// TIA Portal V20 export
FUNCTION "ParameterMove" : Void   // FC22, LAD
// stored: SetENOAutomatically false
   VAR_TEMP
      tempSoftCamDRApplyLoop : Array[1..41] of Int;
      tempSoftCamDRReadLoop : Array[1..41] of Int;
      tempButtonRisingEdge : "HMI_IF_Parameter_Save Button_UDT";
   END_VAR
   VAR_TEMP   // added for the SCL form of the ladder/FBD networks
      _w1 : Bool;
      _w2 : Bool;
      _w3 : Bool;
   END_VAR
BEGIN

REGION Network 2 (SCL): Button Rising Edge
   #tempButtonRisingEdge.Read := "HMI_Interface_Parameter"."Save Button".Read AND NOT "HMI_Interface_Parameter"."Save Button Old".Read;
   #tempButtonRisingEdge.Save := "HMI_Interface_Parameter"."Save Button".Save AND NOT "HMI_Interface_Parameter"."Save Button Old".Save;
   #tempButtonRisingEdge.Apply := "HMI_Interface_Parameter"."Save Button".Apply AND NOT "HMI_Interface_Parameter"."Save Button Old".Apply;
   "HMI_Interface_Parameter"."Save Button Old".Read := "HMI_Interface_Parameter"."Save Button".Read;
   "HMI_Interface_Parameter"."Save Button Old".Save := "HMI_Interface_Parameter"."Save Button".Save;
   "HMI_Interface_Parameter"."Save Button Old".Apply := "HMI_Interface_Parameter"."Save Button".Apply;
END_REGION

REGION Network 3 (SCL): HMI Parameter Text Set Value
   IF #tempButtonRisingEdge.Apply THEN
       "HMI_Interface_Parameter".Parameter_Text[0]."Process Value" := "HMI_Interface_Parameter".Parameter_Text[0]."Set Value";
       "HMI_Interface_Parameter".Parameter_Text[2]."Process Value" := "HMI_Interface_Parameter".Parameter_Text[2]."Set Value";
       "HMI_Interface_Parameter".Parameter_Text[6]."Process Value" := "HMI_Interface_Parameter".Parameter_Text[6]."Set Value";
       "HMI_Interface_Parameter".Parameter_Text[7]."Process Value" := "HMI_Interface_Parameter".Parameter_Text[7]."Set Value";
       "HMI_Interface_Parameter".Parameter_Text[9]."Process Value" := "HMI_Interface_Parameter".Parameter_Text[9]."Set Value";
       "HMI_Interface_Parameter".Parameter_Text[10]."Process Value" := "HMI_Interface_Parameter".Parameter_Text[10]."Set Value";
       "HMI_Interface_Parameter".Parameter_Text[11]."Process Value" := "HMI_Interface_Parameter".Parameter_Text[11]."Set Value";
       "HMI_Interface_Parameter".Parameter_Text[13]."Process Value" := "HMI_Interface_Parameter".Parameter_Text[13]."Set Value";
       "HMI_Interface_Parameter".Parameter_Text[14]."Process Value" := "HMI_Interface_Parameter".Parameter_Text[14]."Set Value";
       "HMI_Interface_Parameter".Parameter_Text[15]."Process Value" := "HMI_Interface_Parameter".Parameter_Text[15]."Set Value";
       "HMI_Interface_Parameter".Parameter_Text[16]."Process Value" := "HMI_Interface_Parameter".Parameter_Text[16]."Set Value";
       "HMI_Interface_Parameter".Parameter_Text[17]."Process Value" := "HMI_Interface_Parameter".Parameter_Text[17]."Set Value";
       "HMI_Interface_Parameter".Parameter_Text[18]."Process Value" := "HMI_Interface_Parameter".Parameter_Text[18]."Set Value";
       "HMI_Interface_Parameter".Parameter_Text[19]."Process Value" := "HMI_Interface_Parameter".Parameter_Text[19]."Set Value";
       "HMI_Interface_Parameter".Parameter_Text[20]."Process Value" := "HMI_Interface_Parameter".Parameter_Text[20]."Set Value";
       "HMI_Interface_Parameter".Parameter_Text[21]."Process Value" := "HMI_Interface_Parameter".Parameter_Text[21]."Set Value";
       "HMI_Interface_Parameter".Parameter_Text[22]."Process Value" := "HMI_Interface_Parameter".Parameter_Text[22]."Set Value";
       "HMI_Interface_Parameter".Parameter_Text[23]."Process Value" := "HMI_Interface_Parameter".Parameter_Text[23]."Set Value";
       "HMI_Interface_Parameter".Parameter_Text[24]."Process Value" := "HMI_Interface_Parameter".Parameter_Text[24]."Set Value";
       "HMI_Interface_Parameter".Parameter_Text[25]."Process Value" := "HMI_Interface_Parameter".Parameter_Text[25]."Set Value";
       "HMI_Interface_Parameter".Parameter_Text[26]."Process Value" := "HMI_Interface_Parameter".Parameter_Text[26]."Set Value";
       "HMI_Interface_Parameter".Parameter_Text[27]."Process Value" := "HMI_Interface_Parameter".Parameter_Text[27]."Set Value";
       "HMI_Interface_Parameter".Parameter_Text[28]."Process Value" := "HMI_Interface_Parameter".Parameter_Text[28]."Set Value";
       "HMI_Interface_Parameter".Parameter_Text[29]."Process Value" := "HMI_Interface_Parameter".Parameter_Text[29]."Set Value";
       "HMI_Interface_Parameter".Parameter_Text[30]."Process Value" := "HMI_Interface_Parameter".Parameter_Text[30]."Set Value";
       "HMI_Interface_Parameter".Parameter_Text[31]."Process Value" := "HMI_Interface_Parameter".Parameter_Text[31]."Set Value";
       "HMI_Interface_Parameter".Parameter_Text[32]."Process Value" := "HMI_Interface_Parameter".Parameter_Text[32]."Set Value";
       "HMI_Interface_Parameter".Parameter_Text[33]."Process Value" := "HMI_Interface_Parameter".Parameter_Text[33]."Set Value";
       "HMI_Interface_Parameter".Parameter_Text[34]."Process Value" := "HMI_Interface_Parameter".Parameter_Text[34]."Set Value";
       "HMI_Interface_Parameter".Parameter_Text[35]."Process Value" := "HMI_Interface_Parameter".Parameter_Text[35]."Set Value";
       "HMI_Interface_Parameter".Parameter_Text[36]."Process Value" := "HMI_Interface_Parameter".Parameter_Text[36]."Set Value";
       "HMI_Interface_Parameter".Parameter_Text[37]."Process Value" := "HMI_Interface_Parameter".Parameter_Text[37]."Set Value";
       "HMI_Interface_Parameter".Parameter_Text[38]."Process Value" := "HMI_Interface_Parameter".Parameter_Text[38]."Set Value";
       "HMI_Interface_Parameter".Parameter_Text[39]."Process Value" := "HMI_Interface_Parameter".Parameter_Text[39]."Set Value";
       "HMI_Interface_Parameter".Parameter_Text[40]."Process Value" := "HMI_Interface_Parameter".Parameter_Text[40]."Set Value";
       "HMI_Interface_Parameter".Parameter_Text[41]."Process Value" := "HMI_Interface_Parameter".Parameter_Text[41]."Set Value";
       "HMI_Interface_Parameter".Parameter_Text[42]."Process Value" := "HMI_Interface_Parameter".Parameter_Text[42]."Set Value";
       "HMI_Interface_Parameter".Parameter_Text[43]."Process Value" := "HMI_Interface_Parameter".Parameter_Text[43]."Set Value";
       "HMI_Interface_Parameter".Parameter_Text[44]."Process Value" := "HMI_Interface_Parameter".Parameter_Text[44]."Set Value";
       "HMI_Interface_Parameter".Parameter_Text[45]."Process Value" := "HMI_Interface_Parameter".Parameter_Text[45]."Set Value";
       "HMI_Interface_Parameter".Parameter_Text[46]."Process Value" := "HMI_Interface_Parameter".Parameter_Text[46]."Set Value";
       "HMI_Interface_Parameter".Parameter_Text[47]."Process Value" := "HMI_Interface_Parameter".Parameter_Text[47]."Set Value";
       "HMI_Interface_Parameter".Parameter_Text[48]."Process Value" := "HMI_Interface_Parameter".Parameter_Text[48]."Set Value";
       "HMI_Interface_Parameter".Parameter_Text[49]."Process Value" := "HMI_Interface_Parameter".Parameter_Text[49]."Set Value";
       "HMI_Interface_Parameter".Parameter_Text[50]."Process Value" := "HMI_Interface_Parameter".Parameter_Text[50]."Set Value";
       "HMI_Interface_Parameter".Parameter_Text[51]."Process Value" := "HMI_Interface_Parameter".Parameter_Text[51]."Set Value";
       "HMI_Interface_Parameter".Parameter_Text[52]."Process Value" := "HMI_Interface_Parameter".Parameter_Text[52]."Set Value";
       "HMI_Interface_Parameter".Parameter_Text[53]."Process Value" := "HMI_Interface_Parameter".Parameter_Text[53]."Set Value";
       "HMI_Interface_Parameter".Parameter_Text[54]."Process Value" := "HMI_Interface_Parameter".Parameter_Text[54]."Set Value";
       "HMI_Interface_Parameter".Parameter_Text[55]."Process Value" := "HMI_Interface_Parameter".Parameter_Text[55]."Set Value";
       "HMI_Interface_Parameter".Parameter_Text[56]."Process Value" := "HMI_Interface_Parameter".Parameter_Text[56]."Set Value";
       "HMI_Interface_Parameter".Parameter_Text[57]."Process Value" := "HMI_Interface_Parameter".Parameter_Text[57]."Set Value";
       "HMI_Interface_Parameter".Parameter_Text[58]."Process Value" := "HMI_Interface_Parameter".Parameter_Text[58]."Set Value";
       "HMI_Interface_Parameter".Parameter_Text[59]."Process Value" := "HMI_Interface_Parameter".Parameter_Text[59]."Set Value";
       "HMI_Interface_Parameter".Parameter_Text[60]."Process Value" := "HMI_Interface_Parameter".Parameter_Text[60]."Set Value";
       "HMI_Interface_Parameter".Parameter_Text[61]."Process Value" := "HMI_Interface_Parameter".Parameter_Text[61]."Set Value";
       "HMI_Interface_Parameter".Parameter_Text[62]."Process Value" := "HMI_Interface_Parameter".Parameter_Text[62]."Set Value";
       "HMI_Interface_Parameter".Parameter_Text[63]."Process Value" := "HMI_Interface_Parameter".Parameter_Text[63]."Set Value";
       "HMI_Interface_Parameter".Parameter_Text[64]."Process Value" := "HMI_Interface_Parameter".Parameter_Text[64]."Set Value";
       "HMI_Interface_Parameter".Parameter_Text[65]."Process Value" := "HMI_Interface_Parameter".Parameter_Text[65]."Set Value";
       "HMI_Interface_Parameter".Parameter_Text[66]."Process Value" := "HMI_Interface_Parameter".Parameter_Text[66]."Set Value";
       "HMI_Interface_Parameter".Parameter_Text[67]."Process Value" := "HMI_Interface_Parameter".Parameter_Text[67]."Set Value";
       "HMI_Interface_Parameter".Parameter_Text[68]."Process Value" := "HMI_Interface_Parameter".Parameter_Text[68]."Set Value";
       "HMI_Interface_Parameter".Parameter_Text[69]."Process Value" := "HMI_Interface_Parameter".Parameter_Text[69]."Set Value";
       "HMI_Interface_Parameter".Parameter_Text[70]."Process Value" := "HMI_Interface_Parameter".Parameter_Text[70]."Set Value";
       "HMI_Interface_Parameter".Parameter_Text[71]."Process Value" := "HMI_Interface_Parameter".Parameter_Text[71]."Set Value";
       "HMI_Interface_Parameter".Parameter_Text[72]."Process Value" := "HMI_Interface_Parameter".Parameter_Text[72]."Set Value";
       "HMI_Interface_Parameter".Parameter_Text[73]."Process Value" := "HMI_Interface_Parameter".Parameter_Text[73]."Set Value";
       "HMI_Interface_Parameter".Parameter_Text[74]."Process Value" := "HMI_Interface_Parameter".Parameter_Text[74]."Set Value";
       "HMI_Interface_Parameter".Parameter_Text[75]."Process Value" := "HMI_Interface_Parameter".Parameter_Text[75]."Set Value";
       "HMI_Interface_Parameter".Parameter_Text[76]."Process Value" := "HMI_Interface_Parameter".Parameter_Text[76]."Set Value";
       "HMI_Interface_Parameter".Parameter_Text[77]."Process Value" := "HMI_Interface_Parameter".Parameter_Text[77]."Set Value";
       "HMI_Interface_Parameter".Parameter_Text[78]."Process Value" := "HMI_Interface_Parameter".Parameter_Text[78]."Set Value";
       "HMI_Interface_Parameter".Parameter_Text[79]."Process Value" := "HMI_Interface_Parameter".Parameter_Text[79]."Set Value";
       "HMI_Interface_Parameter".Parameter_Text[80]."Process Value" := "HMI_Interface_Parameter".Parameter_Text[80]."Set Value";
       "HMI_Interface_Parameter".Parameter_Text[81]."Process Value" := "HMI_Interface_Parameter".Parameter_Text[81]."Set Value";
       "HMI_Interface_Parameter".Parameter_Text[82]."Process Value" := "HMI_Interface_Parameter".Parameter_Text[82]."Set Value";
       "HMI_Interface_Parameter".Parameter_Text[83]."Process Value" := "HMI_Interface_Parameter".Parameter_Text[83]."Set Value";
       "HMI_Interface_Parameter".Parameter_Text[84]."Process Value" := "HMI_Interface_Parameter".Parameter_Text[84]."Set Value";
       "HMI_Interface_Parameter".Parameter_Text[85]."Process Value" := "HMI_Interface_Parameter".Parameter_Text[85]."Set Value";
       "HMI_Interface_Parameter".Parameter_Text[86]."Process Value" := "HMI_Interface_Parameter".Parameter_Text[86]."Set Value";
       "HMI_Interface_Parameter".Parameter_Text[87]."Process Value" := "HMI_Interface_Parameter".Parameter_Text[87]."Set Value";
       "HMI_Interface_Parameter".Parameter_Text[88]."Process Value" := "HMI_Interface_Parameter".Parameter_Text[88]."Set Value";
       "HMI_Interface_Parameter".Parameter_Text[89]."Process Value" := "HMI_Interface_Parameter".Parameter_Text[89]."Set Value";
       "HMI_Interface_Parameter".Parameter_Text[90]."Process Value" := "HMI_Interface_Parameter".Parameter_Text[90]."Set Value";
       "HMI_Interface_Parameter".Parameter_Text[91]."Process Value" := "HMI_Interface_Parameter".Parameter_Text[91]."Set Value";
       "HMI_Interface_Parameter".Parameter_Text[92]."Process Value" := "HMI_Interface_Parameter".Parameter_Text[92]."Set Value";
       "HMI_Interface_Parameter".Parameter_Text[93]."Process Value" := "HMI_Interface_Parameter".Parameter_Text[93]."Set Value";
       "HMI_Interface_Parameter".Parameter_Text[94]."Process Value" := "HMI_Interface_Parameter".Parameter_Text[94]."Set Value";
       "HMI_Interface_Parameter".Parameter_Text[95]."Process Value" := "HMI_Interface_Parameter".Parameter_Text[95]."Set Value";
       "HMI_Interface_Parameter".Parameter_Text[96]."Process Value" := "HMI_Interface_Parameter".Parameter_Text[96]."Set Value";
       "HMI_Interface_Parameter".Parameter_Text[97]."Process Value" := "HMI_Interface_Parameter".Parameter_Text[97]."Set Value";
       "HMI_Interface_Parameter".Parameter_Text[98]."Process Value" := "HMI_Interface_Parameter".Parameter_Text[98]."Set Value";
       "HMI_Interface_Parameter".Parameter_Text[99]."Process Value" := "HMI_Interface_Parameter".Parameter_Text[99]."Set Value";
       "HMI_Interface_Parameter".Parameter_Text[100]."Process Value" := "HMI_Interface_Parameter".Parameter_Text[100]."Set Value";
       "HMI_Interface_Parameter".Parameter_Text[101]."Process Value" := "HMI_Interface_Parameter".Parameter_Text[101]."Set Value";
       "HMI_Interface_Parameter".Parameter_Text[102]."Process Value" := "HMI_Interface_Parameter".Parameter_Text[102]."Set Value";
       "HMI_Interface_Parameter".Parameter_Text[103]."Process Value" := "HMI_Interface_Parameter".Parameter_Text[103]."Set Value";
       "HMI_Interface_Parameter".Parameter_Text[104]."Process Value" := "HMI_Interface_Parameter".Parameter_Text[104]."Set Value";
       "HMI_Interface_Parameter".Parameter_Text[105]."Process Value" := "HMI_Interface_Parameter".Parameter_Text[105]."Set Value";
       "HMI_Interface_Parameter".Parameter_Text[106]."Process Value" := "HMI_Interface_Parameter".Parameter_Text[106]."Set Value";
       "HMI_Interface_Parameter".Parameter_Text[107]."Process Value" := "HMI_Interface_Parameter".Parameter_Text[107]."Set Value";
       "HMI_Interface_Parameter".Parameter_Text[108]."Process Value" := "HMI_Interface_Parameter".Parameter_Text[108]."Set Value";
       "HMI_Interface_Parameter".Parameter_Text[109]."Process Value" := "HMI_Interface_Parameter".Parameter_Text[109]."Set Value";
       "HMI_Interface_Parameter".Parameter_Text[110]."Process Value" := "HMI_Interface_Parameter".Parameter_Text[110]."Set Value";
       "HMI_Interface_Parameter".Parameter_Text[111]."Process Value" := "HMI_Interface_Parameter".Parameter_Text[111]."Set Value";
       "HMI_Interface_Parameter".Parameter_Text[112]."Process Value" := "HMI_Interface_Parameter".Parameter_Text[112]."Set Value";
       "HMI_Interface_Parameter".Parameter_Text[113]."Process Value" := "HMI_Interface_Parameter".Parameter_Text[113]."Set Value";
       "HMI_Interface_Parameter".Parameter_Text[114]."Process Value" := "HMI_Interface_Parameter".Parameter_Text[114]."Set Value";
       "HMI_Interface_Parameter".Parameter_Text[115]."Process Value" := "HMI_Interface_Parameter".Parameter_Text[115]."Set Value";
       "HMI_Interface_Parameter".Parameter_Text[116]."Process Value" := "HMI_Interface_Parameter".Parameter_Text[116]."Set Value";
       "HMI_Interface_Parameter".Parameter_Text[117]."Process Value" := "HMI_Interface_Parameter".Parameter_Text[117]."Set Value";
       "HMI_Interface_Parameter".Parameter_Text[118]."Process Value" := "HMI_Interface_Parameter".Parameter_Text[118]."Set Value";
       "HMI_Interface_Parameter".Parameter_Text[119]."Process Value" := "HMI_Interface_Parameter".Parameter_Text[119]."Set Value";
       "HMI_Interface_Parameter".Parameter_Text[120]."Process Value" := "HMI_Interface_Parameter".Parameter_Text[120]."Set Value";
       "HMI_Interface_Parameter".Parameter_Text[121]."Process Value" := "HMI_Interface_Parameter".Parameter_Text[121]."Set Value";
       "HMI_Interface_Parameter".Parameter_Text[122]."Process Value" := "HMI_Interface_Parameter".Parameter_Text[122]."Set Value";
       "HMI_Interface_Parameter".Parameter_Text[123]."Process Value" := "HMI_Interface_Parameter".Parameter_Text[123]."Set Value";
       "HMI_Interface_Parameter".Parameter_Text[124]."Process Value" := "HMI_Interface_Parameter".Parameter_Text[124]."Set Value";
       "HMI_Interface_Parameter".Parameter_Text[125]."Process Value" := "HMI_Interface_Parameter".Parameter_Text[125]."Set Value";
       "HMI_Interface_Parameter".Parameter_Text[126]."Process Value" := "HMI_Interface_Parameter".Parameter_Text[126]."Set Value";
       "HMI_Interface_Parameter".Parameter_Text[127]."Process Value" := "HMI_Interface_Parameter".Parameter_Text[127]."Set Value";
       "HMI_Interface_Parameter".Parameter_Text[128]."Process Value" := "HMI_Interface_Parameter".Parameter_Text[128]."Set Value";
       "HMI_Interface_Parameter".Parameter_Text[129]."Process Value" := "HMI_Interface_Parameter".Parameter_Text[129]."Set Value";
       "HMI_Interface_Parameter".Parameter_Text[130]."Process Value" := "HMI_Interface_Parameter".Parameter_Text[130]."Set Value";
       "HMI_Interface_Parameter".Parameter_Text[131]."Process Value" := "HMI_Interface_Parameter".Parameter_Text[131]."Set Value";
       "HMI_Interface_Parameter".Parameter_Text[132]."Process Value" := "HMI_Interface_Parameter".Parameter_Text[132]."Set Value";
       "HMI_Interface_Parameter".Parameter_Text[133]."Process Value" := "HMI_Interface_Parameter".Parameter_Text[133]."Set Value";
       "HMI_Interface_Parameter".Parameter_Text[134]."Process Value" := "HMI_Interface_Parameter".Parameter_Text[134]."Set Value";
       "HMI_Interface_Parameter".Parameter_Text[135]."Process Value" := "HMI_Interface_Parameter".Parameter_Text[135]."Set Value";
       "HMI_Interface_Parameter".Parameter_Text[136]."Process Value" := "HMI_Interface_Parameter".Parameter_Text[136]."Set Value";
       "HMI_Interface_Parameter".Parameter_Text[137]."Process Value" := "HMI_Interface_Parameter".Parameter_Text[137]."Set Value";
       "HMI_Interface_Parameter".Parameter_Text[138]."Process Value" := "HMI_Interface_Parameter".Parameter_Text[138]."Set Value";
       "HMI_Interface_Parameter".Parameter_Text[139]."Process Value" := "HMI_Interface_Parameter".Parameter_Text[139]."Set Value";
       "HMI_Interface_Parameter".Parameter_Text[140]."Process Value" := "HMI_Interface_Parameter".Parameter_Text[140]."Set Value";
       "HMI_Interface_Parameter".Parameter_Text[141]."Process Value" := "HMI_Interface_Parameter".Parameter_Text[141]."Set Value";
       "HMI_Interface_Parameter".Parameter_Text[142]."Process Value" := "HMI_Interface_Parameter".Parameter_Text[142]."Set Value";
       "HMI_Interface_Parameter".Parameter_Text[143]."Process Value" := "HMI_Interface_Parameter".Parameter_Text[143]."Set Value";
       "HMI_Interface_Parameter".Parameter_Text[144]."Process Value" := "HMI_Interface_Parameter".Parameter_Text[144]."Set Value";
       "HMI_Interface_Parameter".Parameter_Text[145]."Process Value" := "HMI_Interface_Parameter".Parameter_Text[145]."Set Value";
       "HMI_Interface_Parameter".Parameter_Text[146]."Process Value" := "HMI_Interface_Parameter".Parameter_Text[146]."Set Value";
       "HMI_Interface_Parameter".Parameter_Text[147]."Process Value" := "HMI_Interface_Parameter".Parameter_Text[147]."Set Value";
       "HMI_Interface_Parameter".Parameter_Text[148]."Process Value" := "HMI_Interface_Parameter".Parameter_Text[148]."Set Value";
       "HMI_Interface_Parameter".Parameter_Text[149]."Process Value" := "HMI_Interface_Parameter".Parameter_Text[149]."Set Value";
       "HMI_Interface_Parameter".Parameter_Text[150]."Process Value" := "HMI_Interface_Parameter".Parameter_Text[150]."Set Value";
       "HMI_Interface_Parameter".Parameter_Text[151]."Process Value" := "HMI_Interface_Parameter".Parameter_Text[151]."Set Value";
       "HMI_Interface_Parameter".Parameter_Text[152]."Process Value" := "HMI_Interface_Parameter".Parameter_Text[152]."Set Value";
       "HMI_Interface_Parameter".Parameter_Text[153]."Process Value" := "HMI_Interface_Parameter".Parameter_Text[153]."Set Value";
       "HMI_Interface_Parameter".Parameter_Text[154]."Process Value" := "HMI_Interface_Parameter".Parameter_Text[154]."Set Value";
   END_IF;
END_REGION

REGION Network 4 (SCL): HMI Parameter Image Set Value
   IF #tempButtonRisingEdge.Apply THEN
       // Move to recipe (Network 7)
       (* Unit1.Em3.HmiInterface.auxiliary.dancerRegulator := "HMI_Interface_Parameter".Parameter_Image[0]."Set Value";
       Unit1.Em0.HmiInterface.auxiliary.AutoSpliceRemainingLength := "HMI_Interface_Parameter".Parameter_Image[1]."Set Value";
       Unit1.Em1.HmiInterface.auxiliary.AutoSpliceRemainingLength := "HMI_Interface_Parameter".Parameter_Image[1]."Set Value"; *)
       "HMI_Interface_Parameter".FATModeInterface.HoursTest.ProcessValue.SelectHours_ProcessValue := "HMI_Interface_Parameter".FATModeInterface.HoursTest.SetValue.SelectHours_SetValue;
       "HMI_Interface_Parameter".FATModeInterface.Sampling.ProcessValue.SelectCount_ProcessValue := "HMI_Interface_Parameter".FATModeInterface.Sampling.SetValue.SelectCount_SetValue;
   END_IF;
   //
   //
   "Unit1.EmNodes".FATModeInterface.HoursTest.ProcessValue.SelectHours_ProcessValue := "HMI_Interface_Parameter".FATModeInterface.HoursTest.SetValue.SelectHours_SetValue;
   "Unit1.EmNodes".FATModeInterface.Sampling.ProcessValue.SelectCount_ProcessValue := "HMI_Interface_Parameter".FATModeInterface.Sampling.SetValue.SelectCount_SetValue;

   "HMI_Interface_Parameter".FATModeInterface.Capability.ProcessValue.CapabilityCount := LREAL_TO_INT("Unit1.EmNodes".BA060.InspectionToStack.InterfaceData.LReal[14]);
   "HMI_Interface_Parameter".FATModeInterface.Capability.ProcessValue.SelectCycle_ProcessValue := LREAL_TO_INT("Unit1.EmNodes".BA060.InspectionToStack.InterfaceData.LReal[15]);
   "HMI_Interface_Parameter".FATModeInterface.Capability.SetValue.SelectCycle_SetValue := LREAL_TO_INT("Unit1.EmNodes".BA060.InspectionToStack.InterfaceData.LReal[15]);


   "Unit1.EmNodes".FATModeInterface.Capability.ProcessValue.CapabilityCount := LREAL_TO_INT("Unit1.EmNodes".BA060.InspectionToStack.InterfaceData.LReal[14]);
   "Unit1.EmNodes".FATModeInterface.Capability.ProcessValue.SelectCycle_ProcessValue := LREAL_TO_INT("Unit1.EmNodes".BA060.InspectionToStack.InterfaceData.LReal[15]);
END_REGION

REGION Network 5 (SCL): HMI Parameter Text Process Value
   "Unit1.MotionNodes".PLCToMotion.Parameters.StackMain.Global.CPM := "HMI_Interface_Parameter".Parameter_Text[0]."Process Value";
   // FFU (Motion 소스 없음)
   // Unit1.MotionNodes.PLCToMotion.Parameters.StackMain.Auto.CellCount := LREAL_TO_DINT("HMI_Interface_Parameter".Parameter_Text[2]."Process Value");
   // JR Winding Turn Count (Motion 소스 없음)
   // Top Unwinder Bobin Size (Motion 소스 없음)
   // Bottom Unwinder Bobin Size (Motion 소스 없음)
   "Unit1.EmNodes".SleepModeActivationTime := DINT_TO_TIME(ROUND("HMI_Interface_Parameter".Parameter_Text[6]."Process Value" * 1000));
   "Unit1.EmNodes".DeepSleepModeActivationTime := DINT_TO_TIME(ROUND("HMI_Interface_Parameter".Parameter_Text[7]."Process Value" * 1000));
   // Reserve9 (Motion 소스 없음)
   "Unit1.MotionNodes".PLCToMotion.Parameters.Dancer.Setpoint := "HMI_Interface_Parameter".Parameter_Text[9]."Process Value";
   "Unit1.MotionNodes".PLCToMotion.Parameters.Dancer.Kp := "HMI_Interface_Parameter".Parameter_Text[10]."Process Value";
   "Unit1.MotionNodes".PLCToMotion.Parameters.Dancer.Ki := "HMI_Interface_Parameter".Parameter_Text[11]."Process Value";
   "Unit1.MotionNodes".PLCToMotion.Parameters.StackMain.Global.StageWidth := "HMI_Interface_Parameter".Parameter_Text[12]."Process Value";
   "Unit1.MotionNodes".PLCToMotion.Parameters.StackMain.Auto.Pos1FinalRollerXFwdOutputCam := "HMI_Interface_Parameter".Parameter_Text[13]."Process Value";
   "Unit1.MotionNodes".PLCToMotion.Parameters.StackMain.Auto.Pos1FinalRollerXBwdOutputCam := "HMI_Interface_Parameter".Parameter_Text[14]."Process Value";
   "Unit1.MotionNodes".PLCToMotion.Parameters.StackMain.Auto.Pos1FinalRollerXStackTableDownOutputCam := "HMI_Interface_Parameter".Parameter_Text[15]."Process Value";
   "Unit1.MotionNodes".PLCToMotion.Parameters.StackMain.Auto.Pos1FinalRollerXStackAnodeVisionOutputCam := "HMI_Interface_Parameter".Parameter_Text[16]."Process Value";
   "Unit1.MotionNodes".PLCToMotion.Parameters.StackMain.Auto.Pos1FinalRollerXStackCathodeVisionOutputCam := "HMI_Interface_Parameter".Parameter_Text[17]."Process Value";
   "Unit1.MotionNodes".PLCToMotion.Parameters.StackMain.Auto.Pos1AnodePnPX1FwdOutputCam := "HMI_Interface_Parameter".Parameter_Text[18]."Process Value";
   "Unit1.MotionNodes".PLCToMotion.Parameters.StackMain.Auto.Pos1AnodePnPX1BwdOutputCam := "HMI_Interface_Parameter".Parameter_Text[19]."Process Value";
   "Unit1.MotionNodes".PLCToMotion.Parameters.StackMain.Auto.Pos1AnodePnPX1ReelCutDataDeleteOffOutputCam := "HMI_Interface_Parameter".Parameter_Text[20]."Process Value";
   "Unit1.MotionNodes".PLCToMotion.Parameters.StackMain.Auto.Pos1AnodePnPX2FwdOutputCam := "HMI_Interface_Parameter".Parameter_Text[21]."Process Value";
   "Unit1.MotionNodes".PLCToMotion.Parameters.StackMain.Auto.Pos1AnodePnPX2BwdOutputCam := "HMI_Interface_Parameter".Parameter_Text[22]."Process Value";
   "Unit1.MotionNodes".PLCToMotion.Parameters.StackMain.Auto.Pos1AnodePnPZ1Down1OutputCam := "HMI_Interface_Parameter".Parameter_Text[23]."Process Value";
   "Unit1.MotionNodes".PLCToMotion.Parameters.StackMain.Auto.Pos1AnodePnPZ1Up1OutputCam := "HMI_Interface_Parameter".Parameter_Text[24]."Process Value";
   "Unit1.MotionNodes".PLCToMotion.Parameters.StackMain.Auto.Pos1AnodePnPZ2Down1OutputCam := "HMI_Interface_Parameter".Parameter_Text[25]."Process Value";
   "Unit1.MotionNodes".PLCToMotion.Parameters.StackMain.Auto.Pos1AnodePnPZ2Up1OutputCam := "HMI_Interface_Parameter".Parameter_Text[26]."Process Value";
   "Unit1.MotionNodes".PLCToMotion.Parameters.StackMain.Auto.Pos1AnodePnPZ1Down2OutputCam := "HMI_Interface_Parameter".Parameter_Text[27]."Process Value";
   "Unit1.MotionNodes".PLCToMotion.Parameters.StackMain.Auto.Pos1AnodePnPZ1Up2OutputCam := "HMI_Interface_Parameter".Parameter_Text[28]."Process Value";
   "Unit1.MotionNodes".PLCToMotion.Parameters.StackMain.Auto.Pos1AnodePnPZ2Down2OutputCam := "HMI_Interface_Parameter".Parameter_Text[29]."Process Value";
   "Unit1.MotionNodes".PLCToMotion.Parameters.StackMain.Auto.Pos1AnodePnPZ2Up2OutputCam := "HMI_Interface_Parameter".Parameter_Text[30]."Process Value";
   "Unit1.MotionNodes".PLCToMotion.Parameters.StackMain.Auto.Pos1AnodePnPZ1SuctionOnOutputCam := "HMI_Interface_Parameter".Parameter_Text[31]."Process Value";
   "Unit1.MotionNodes".PLCToMotion.Parameters.StackMain.Auto.Pos1AnodePnPZ1SuctionOffOutputCam := "HMI_Interface_Parameter".Parameter_Text[32]."Process Value";
   "Unit1.MotionNodes".PLCToMotion.Parameters.StackMain.Auto.Pos1AnodePnPZ1ReelCutBlowOutputCam := "HMI_Interface_Parameter".Parameter_Text[33]."Process Value";
   "Unit1.MotionNodes".PLCToMotion.Parameters.StackMain.Auto.Pos1AnodePnPZ1ReelCutDataDeleteOnOutputCam := "HMI_Interface_Parameter".Parameter_Text[34]."Process Value";
   "Unit1.MotionNodes".PLCToMotion.Parameters.StackMain.Auto.Pos1AnodePnPZ1AlignVisionOutputCam := "HMI_Interface_Parameter".Parameter_Text[35]."Process Value";
   "Unit1.MotionNodes".PLCToMotion.Parameters.StackMain.Auto.Pos1AnodePnPZ2SuctionOnOutputCam := "HMI_Interface_Parameter".Parameter_Text[36]."Process Value";
   "Unit1.MotionNodes".PLCToMotion.Parameters.StackMain.Auto.Pos1AnodePnPZ2SuctionOffOutputCam := "HMI_Interface_Parameter".Parameter_Text[37]."Process Value";
   "Unit1.MotionNodes".PLCToMotion.Parameters.StackMain.Auto.Pos1AnodeAlignSuctionOnOutputCam := "HMI_Interface_Parameter".Parameter_Text[38]."Process Value";
   "Unit1.MotionNodes".PLCToMotion.Parameters.StackMain.Auto.Pos1AnodeAlignSuctionOffOutputCam := "HMI_Interface_Parameter".Parameter_Text[39]."Process Value";
   "Unit1.MotionNodes".PLCToMotion.Parameters.StackMain.Auto.Pos1CathodePnPX1FwdOutputCam := "HMI_Interface_Parameter".Parameter_Text[40]."Process Value";
   "Unit1.MotionNodes".PLCToMotion.Parameters.StackMain.Auto.Pos1CathodePnPX1BwdOutputCam := "HMI_Interface_Parameter".Parameter_Text[41]."Process Value";
   "Unit1.MotionNodes".PLCToMotion.Parameters.StackMain.Auto.Pos1CathodePnPX1ReelCutDataDeleteOffOutputCam := "HMI_Interface_Parameter".Parameter_Text[42]."Process Value";
   "Unit1.MotionNodes".PLCToMotion.Parameters.StackMain.Auto.Pos1CathodePnPX2FwdOutputCam := "HMI_Interface_Parameter".Parameter_Text[43]."Process Value";
   "Unit1.MotionNodes".PLCToMotion.Parameters.StackMain.Auto.Pos1CathodePnPX2BwdOutputCam := "HMI_Interface_Parameter".Parameter_Text[44]."Process Value";
   "Unit1.MotionNodes".PLCToMotion.Parameters.StackMain.Auto.Pos1CathodePnPZ1Down1OutputCam := "HMI_Interface_Parameter".Parameter_Text[45]."Process Value";
   "Unit1.MotionNodes".PLCToMotion.Parameters.StackMain.Auto.Pos1CathodePnPZ1Up1OutputCam := "HMI_Interface_Parameter".Parameter_Text[46]."Process Value";
   "Unit1.MotionNodes".PLCToMotion.Parameters.StackMain.Auto.Pos1CathodePnPZ2Down1OutputCam := "HMI_Interface_Parameter".Parameter_Text[47]."Process Value";
   "Unit1.MotionNodes".PLCToMotion.Parameters.StackMain.Auto.Pos1CathodePnPZ2Up1OutputCam := "HMI_Interface_Parameter".Parameter_Text[48]."Process Value";
   "Unit1.MotionNodes".PLCToMotion.Parameters.StackMain.Auto.Pos1CathodePnPZ1Down2OutputCam := "HMI_Interface_Parameter".Parameter_Text[49]."Process Value";
   "Unit1.MotionNodes".PLCToMotion.Parameters.StackMain.Auto.Pos1CathodePnPZ1Up2OutputCam := "HMI_Interface_Parameter".Parameter_Text[50]."Process Value";
   "Unit1.MotionNodes".PLCToMotion.Parameters.StackMain.Auto.Pos1CathodePnPZ2Down2OutputCam := "HMI_Interface_Parameter".Parameter_Text[51]."Process Value";
   "Unit1.MotionNodes".PLCToMotion.Parameters.StackMain.Auto.Pos1CathodePnPZ2Up2OutputCam := "HMI_Interface_Parameter".Parameter_Text[52]."Process Value";
   "Unit1.MotionNodes".PLCToMotion.Parameters.StackMain.Auto.Pos1CathodePnPZ1SuctionOnOutputCam := "HMI_Interface_Parameter".Parameter_Text[53]."Process Value";
   "Unit1.MotionNodes".PLCToMotion.Parameters.StackMain.Auto.Pos1CathodePnPZ1SuctionOffOutputCam := "HMI_Interface_Parameter".Parameter_Text[54]."Process Value";
   "Unit1.MotionNodes".PLCToMotion.Parameters.StackMain.Auto.Pos1CathodePnPZ1ReelCutBlowOutputCam := "HMI_Interface_Parameter".Parameter_Text[55]."Process Value";
   "Unit1.MotionNodes".PLCToMotion.Parameters.StackMain.Auto.Pos1CathodePnPZ1ReelCutDataDeleteOnOutputCam := "HMI_Interface_Parameter".Parameter_Text[56]."Process Value";
   "Unit1.MotionNodes".PLCToMotion.Parameters.StackMain.Auto.Pos1CathodePnPZ1AlignVisionOutputCam := "HMI_Interface_Parameter".Parameter_Text[57]."Process Value";
   "Unit1.MotionNodes".PLCToMotion.Parameters.StackMain.Auto.Pos1CathodePnPZ2SuctionOnOutputCam := "HMI_Interface_Parameter".Parameter_Text[58]."Process Value";
   "Unit1.MotionNodes".PLCToMotion.Parameters.StackMain.Auto.Pos1CathodePnPZ2SuctionOffOutputCam := "HMI_Interface_Parameter".Parameter_Text[59]."Process Value";
   "Unit1.MotionNodes".PLCToMotion.Parameters.StackMain.Auto.Pos1CathodeAlignSuctionOnOutputCam := "HMI_Interface_Parameter".Parameter_Text[60]."Process Value";
   "Unit1.MotionNodes".PLCToMotion.Parameters.StackMain.Auto.Pos1CathodeAlignSuctionOffOutputCam := "HMI_Interface_Parameter".Parameter_Text[61]."Process Value";
   "Unit1.MotionNodes".PLCToMotion.Parameters.StackMain.Auto.Pos2FinalRollerXFwdOutputCam := "HMI_Interface_Parameter".Parameter_Text[62]."Process Value";
   "Unit1.MotionNodes".PLCToMotion.Parameters.StackMain.Auto.Pos2FinalRollerXBwdOutputCam := "HMI_Interface_Parameter".Parameter_Text[63]."Process Value";
   "Unit1.MotionNodes".PLCToMotion.Parameters.StackMain.Auto.Pos2FinalRollerXStackTableDownOutputCam := "HMI_Interface_Parameter".Parameter_Text[64]."Process Value";
   "Unit1.MotionNodes".PLCToMotion.Parameters.StackMain.Auto.Pos2FinalRollerXStackAnodeVisionOutputCam := "HMI_Interface_Parameter".Parameter_Text[65]."Process Value";
   "Unit1.MotionNodes".PLCToMotion.Parameters.StackMain.Auto.Pos2FinalRollerXStackCathodeVisionOutputCam := "HMI_Interface_Parameter".Parameter_Text[66]."Process Value";
   "Unit1.MotionNodes".PLCToMotion.Parameters.StackMain.Auto.Pos2AnodePnPX1FwdOutputCam := "HMI_Interface_Parameter".Parameter_Text[67]."Process Value";
   "Unit1.MotionNodes".PLCToMotion.Parameters.StackMain.Auto.Pos2AnodePnPX1BwdOutputCam := "HMI_Interface_Parameter".Parameter_Text[68]."Process Value";
   "Unit1.MotionNodes".PLCToMotion.Parameters.StackMain.Auto.Pos2AnodePnPX1ReelCutDataDeleteOffOutputCam := "HMI_Interface_Parameter".Parameter_Text[69]."Process Value";
   "Unit1.MotionNodes".PLCToMotion.Parameters.StackMain.Auto.Pos2AnodePnPX2FwdOutputCam := "HMI_Interface_Parameter".Parameter_Text[70]."Process Value";
   "Unit1.MotionNodes".PLCToMotion.Parameters.StackMain.Auto.Pos2AnodePnPX2BwdOutputCam := "HMI_Interface_Parameter".Parameter_Text[71]."Process Value";
   "Unit1.MotionNodes".PLCToMotion.Parameters.StackMain.Auto.Pos2AnodePnPZ1Down1OutputCam := "HMI_Interface_Parameter".Parameter_Text[72]."Process Value";
   "Unit1.MotionNodes".PLCToMotion.Parameters.StackMain.Auto.Pos2AnodePnPZ1Up1OutputCam := "HMI_Interface_Parameter".Parameter_Text[73]."Process Value";
   "Unit1.MotionNodes".PLCToMotion.Parameters.StackMain.Auto.Pos2AnodePnPZ2Down1OutputCam := "HMI_Interface_Parameter".Parameter_Text[74]."Process Value";
   "Unit1.MotionNodes".PLCToMotion.Parameters.StackMain.Auto.Pos2AnodePnPZ2Up1OutputCam := "HMI_Interface_Parameter".Parameter_Text[75]."Process Value";
   "Unit1.MotionNodes".PLCToMotion.Parameters.StackMain.Auto.Pos2AnodePnPZ1Down2OutputCam := "HMI_Interface_Parameter".Parameter_Text[76]."Process Value";
   "Unit1.MotionNodes".PLCToMotion.Parameters.StackMain.Auto.Pos2AnodePnPZ1Up2OutputCam := "HMI_Interface_Parameter".Parameter_Text[77]."Process Value";
   "Unit1.MotionNodes".PLCToMotion.Parameters.StackMain.Auto.Pos2AnodePnPZ2Down2OutputCam := "HMI_Interface_Parameter".Parameter_Text[78]."Process Value";
   "Unit1.MotionNodes".PLCToMotion.Parameters.StackMain.Auto.Pos2AnodePnPZ2Up2OutputCam := "HMI_Interface_Parameter".Parameter_Text[79]."Process Value";
   "Unit1.MotionNodes".PLCToMotion.Parameters.StackMain.Auto.Pos2AnodePnPZ1SuctionOnOutputCam := "HMI_Interface_Parameter".Parameter_Text[80]."Process Value";
   "Unit1.MotionNodes".PLCToMotion.Parameters.StackMain.Auto.Pos2AnodePnPZ1SuctionOffOutputCam := "HMI_Interface_Parameter".Parameter_Text[81]."Process Value";
   "Unit1.MotionNodes".PLCToMotion.Parameters.StackMain.Auto.Pos2AnodePnPZ1ReelCutBlowOutputCam := "HMI_Interface_Parameter".Parameter_Text[82]."Process Value";
   "Unit1.MotionNodes".PLCToMotion.Parameters.StackMain.Auto.Pos2AnodePnPZ1ReelCutDataDeleteOnOutputCam := "HMI_Interface_Parameter".Parameter_Text[83]."Process Value";
   "Unit1.MotionNodes".PLCToMotion.Parameters.StackMain.Auto.Pos2AnodePnPZ1AlignVisionOutputCam := "HMI_Interface_Parameter".Parameter_Text[84]."Process Value";
   "Unit1.MotionNodes".PLCToMotion.Parameters.StackMain.Auto.Pos2AnodePnPZ2SuctionOnOutputCam := "HMI_Interface_Parameter".Parameter_Text[85]."Process Value";
   "Unit1.MotionNodes".PLCToMotion.Parameters.StackMain.Auto.Pos2AnodePnPZ2SuctionOffOutputCam := "HMI_Interface_Parameter".Parameter_Text[86]."Process Value";
   "Unit1.MotionNodes".PLCToMotion.Parameters.StackMain.Auto.Pos2AnodeAlignSuctionOnOutputCam := "HMI_Interface_Parameter".Parameter_Text[87]."Process Value";
   "Unit1.MotionNodes".PLCToMotion.Parameters.StackMain.Auto.Pos2AnodeAlignSuctionOffOutputCam := "HMI_Interface_Parameter".Parameter_Text[88]."Process Value";
   "Unit1.MotionNodes".PLCToMotion.Parameters.StackMain.Auto.Pos2CathodePnPX1FwdOutputCam := "HMI_Interface_Parameter".Parameter_Text[89]."Process Value";
   "Unit1.MotionNodes".PLCToMotion.Parameters.StackMain.Auto.Pos2CathodePnPX1BwdOutputCam := "HMI_Interface_Parameter".Parameter_Text[90]."Process Value";
   "Unit1.MotionNodes".PLCToMotion.Parameters.StackMain.Auto.Pos2CathodePnPX1ReelCutDataDeleteOffOutputCam := "HMI_Interface_Parameter".Parameter_Text[91]."Process Value";
   "Unit1.MotionNodes".PLCToMotion.Parameters.StackMain.Auto.Pos2CathodePnPX2FwdOutputCam := "HMI_Interface_Parameter".Parameter_Text[92]."Process Value";
   "Unit1.MotionNodes".PLCToMotion.Parameters.StackMain.Auto.Pos2CathodePnPX2BwdOutputCam := "HMI_Interface_Parameter".Parameter_Text[93]."Process Value";
   "Unit1.MotionNodes".PLCToMotion.Parameters.StackMain.Auto.Pos2CathodePnPZ1Down1OutputCam := "HMI_Interface_Parameter".Parameter_Text[94]."Process Value";
   "Unit1.MotionNodes".PLCToMotion.Parameters.StackMain.Auto.Pos2CathodePnPZ1Up1OutputCam := "HMI_Interface_Parameter".Parameter_Text[95]."Process Value";
   "Unit1.MotionNodes".PLCToMotion.Parameters.StackMain.Auto.Pos2CathodePnPZ2Down1OutputCam := "HMI_Interface_Parameter".Parameter_Text[96]."Process Value";
   "Unit1.MotionNodes".PLCToMotion.Parameters.StackMain.Auto.Pos2CathodePnPZ2Up1OutputCam := "HMI_Interface_Parameter".Parameter_Text[97]."Process Value";
   "Unit1.MotionNodes".PLCToMotion.Parameters.StackMain.Auto.Pos2CathodePnPZ1Down2OutputCam := "HMI_Interface_Parameter".Parameter_Text[98]."Process Value";
   "Unit1.MotionNodes".PLCToMotion.Parameters.StackMain.Auto.Pos2CathodePnPZ1Up2OutputCam := "HMI_Interface_Parameter".Parameter_Text[99]."Process Value";
   "Unit1.MotionNodes".PLCToMotion.Parameters.StackMain.Auto.Pos2CathodePnPZ2Down2OutputCam := "HMI_Interface_Parameter".Parameter_Text[100]."Process Value";
   "Unit1.MotionNodes".PLCToMotion.Parameters.StackMain.Auto.Pos2CathodePnPZ2Up2OutputCam := "HMI_Interface_Parameter".Parameter_Text[101]."Process Value";
   "Unit1.MotionNodes".PLCToMotion.Parameters.StackMain.Auto.Pos2CathodePnPZ1SuctionOnOutputCam := "HMI_Interface_Parameter".Parameter_Text[102]."Process Value";
   "Unit1.MotionNodes".PLCToMotion.Parameters.StackMain.Auto.Pos2CathodePnPZ1SuctionOffOutputCam := "HMI_Interface_Parameter".Parameter_Text[103]."Process Value";
   "Unit1.MotionNodes".PLCToMotion.Parameters.StackMain.Auto.Pos2CathodePnPZ1ReelCutBlowOutputCam := "HMI_Interface_Parameter".Parameter_Text[104]."Process Value";
   "Unit1.MotionNodes".PLCToMotion.Parameters.StackMain.Auto.Pos2CathodePnPZ1ReelCutDataDeleteOnOutputCam := "HMI_Interface_Parameter".Parameter_Text[105]."Process Value";
   "Unit1.MotionNodes".PLCToMotion.Parameters.StackMain.Auto.Pos2CathodePnPZ1AlignVisionOutputCam := "HMI_Interface_Parameter".Parameter_Text[106]."Process Value";
   "Unit1.MotionNodes".PLCToMotion.Parameters.StackMain.Auto.Pos2CathodePnPZ2SuctionOnOutputCam := "HMI_Interface_Parameter".Parameter_Text[107]."Process Value";
   "Unit1.MotionNodes".PLCToMotion.Parameters.StackMain.Auto.Pos2CathodePnPZ2SuctionOffOutputCam := "HMI_Interface_Parameter".Parameter_Text[108]."Process Value";
   "Unit1.MotionNodes".PLCToMotion.Parameters.StackMain.Auto.Pos2CathodeAlignSuctionOnOutputCam := "HMI_Interface_Parameter".Parameter_Text[109]."Process Value";
   "Unit1.MotionNodes".PLCToMotion.Parameters.StackMain.Auto.Pos2CathodeAlignSuctionOffOutputCam := "HMI_Interface_Parameter".Parameter_Text[110]."Process Value";
   "Unit1.MotionNodes".PLCToMotion.Parameters.StackMain.StackCalculate.StageHeight := "HMI_Interface_Parameter".Parameter_Text[111]."Process Value";
   "Unit1.MotionNodes".PLCToMotion.Parameters.StackMain.StackCalculate.StageGap := "HMI_Interface_Parameter".Parameter_Text[112]."Process Value";
   "Unit1.MotionNodes".PLCToMotion.Parameters.StackMain.StackCalculate.Ratio.FinalRollerStart := "HMI_Interface_Parameter".Parameter_Text[113]."Process Value";
   "Unit1.MotionNodes".PLCToMotion.Parameters.StackMain.StackCalculate.Ratio.FinalRollerEnd := "HMI_Interface_Parameter".Parameter_Text[114]."Process Value";
   "Unit1.MotionNodes".PLCToMotion.Parameters.StackMain.StackCalculate.Ratio.PnPXStart := "HMI_Interface_Parameter".Parameter_Text[115]."Process Value";
   "Unit1.MotionNodes".PLCToMotion.Parameters.StackMain.StackCalculate.Ratio.PnPXEnd := "HMI_Interface_Parameter".Parameter_Text[116]."Process Value";
   "Unit1.MotionNodes".PLCToMotion.Parameters.StackMain.StackCalculate.Ratio.PnPZDownStart := "HMI_Interface_Parameter".Parameter_Text[117]."Process Value";
   "Unit1.MotionNodes".PLCToMotion.Parameters.StackMain.StackCalculate.Ratio.PnPZDownEnd := "HMI_Interface_Parameter".Parameter_Text[118]."Process Value";
   "Unit1.MotionNodes".PLCToMotion.Parameters.StackMain.StackCalculate.Ratio.PnPZUpStart := "HMI_Interface_Parameter".Parameter_Text[119]."Process Value";
   "Unit1.MotionNodes".PLCToMotion.Parameters.StackMain.StackCalculate.Ratio.PnPZUpEnd := "HMI_Interface_Parameter".Parameter_Text[120]."Process Value";
   "Unit1.MotionNodes".PLCToMotion.Parameters.StackMain.StackCalculate.Ratio.MandrelBwdStart := "HMI_Interface_Parameter".Parameter_Text[121]."Process Value";
   "Unit1.MotionNodes".PLCToMotion.Parameters.StackMain.StackCalculate.Ratio.MandrelBwdEnd := "HMI_Interface_Parameter".Parameter_Text[122]."Process Value";
   "Unit1.MotionNodes".PLCToMotion.Parameters.StackMain.StackCalculate.Ratio.MandrelFwdStart := "HMI_Interface_Parameter".Parameter_Text[123]."Process Value";
   "Unit1.MotionNodes".PLCToMotion.Parameters.StackMain.StackCalculate.Ratio.MandrelFwdEnd := "HMI_Interface_Parameter".Parameter_Text[124]."Process Value";
   "Unit1.MotionNodes".PLCToMotion.Parameters.StackMain.StackCalculate.Ratio.MandrelUpStart1 := "HMI_Interface_Parameter".Parameter_Text[125]."Process Value";
   "Unit1.MotionNodes".PLCToMotion.Parameters.StackMain.StackCalculate.Ratio.MandrelUpEnd1 := "HMI_Interface_Parameter".Parameter_Text[126]."Process Value";
   "Unit1.MotionNodes".PLCToMotion.Parameters.StackMain.StackCalculate.Ratio.MandrelUpStart2 := "HMI_Interface_Parameter".Parameter_Text[127]."Process Value";
   "Unit1.MotionNodes".PLCToMotion.Parameters.StackMain.StackCalculate.Ratio.MandrelUpEnd2 := "HMI_Interface_Parameter".Parameter_Text[128]."Process Value";
   "Unit1.MotionNodes".PLCToMotion.Parameters.StackMain.StackCalculate.Ratio.MandrelDownStart := "HMI_Interface_Parameter".Parameter_Text[129]."Process Value";
   "Unit1.MotionNodes".PLCToMotion.Parameters.StackMain.StackCalculate.Ratio.MandrelDownEnd := "HMI_Interface_Parameter".Parameter_Text[130]."Process Value";
   "Unit1.MotionNodes".PLCToMotion.Parameters.StackMain.StackCalculate.Ratio.MandrelYTerm := "HMI_Interface_Parameter".Parameter_Text[131]."Process Value";
   "Unit1.MotionNodes".PLCToMotion.Parameters.StackMain.StackCalculate.Ratio.MandrelZTerm := "HMI_Interface_Parameter".Parameter_Text[132]."Process Value";
   "Unit1.MotionNodes".PLCToMotion.Parameters.StackMain.StackCalculate.Ratio.MandrelBwdOffset := "HMI_Interface_Parameter".Parameter_Text[133]."Process Value";
   "Unit1.MotionNodes".PLCToMotion.Parameters.StackMain.StackCalculate.Ratio.MandrelFwdOffset := "HMI_Interface_Parameter".Parameter_Text[134]."Process Value";
   "Unit1.MotionNodes".PLCToMotion.Parameters.StackMain.StackCalculate.Time.FinalRollerStart := "HMI_Interface_Parameter".Parameter_Text[135]."Process Value";
   "Unit1.MotionNodes".PLCToMotion.Parameters.StackMain.StackCalculate.Time.FinalRollerEnd := "HMI_Interface_Parameter".Parameter_Text[136]."Process Value";
   "Unit1.MotionNodes".PLCToMotion.Parameters.StackMain.StackCalculate.Time.PnPXStart := "HMI_Interface_Parameter".Parameter_Text[137]."Process Value";
   "Unit1.MotionNodes".PLCToMotion.Parameters.StackMain.StackCalculate.Time.PnPXEnd := "HMI_Interface_Parameter".Parameter_Text[138]."Process Value";
   "Unit1.MotionNodes".PLCToMotion.Parameters.StackMain.StackCalculate.Time.PnPZDownStart := "HMI_Interface_Parameter".Parameter_Text[139]."Process Value";
   "Unit1.MotionNodes".PLCToMotion.Parameters.StackMain.StackCalculate.Time.PnPZDownEnd := "HMI_Interface_Parameter".Parameter_Text[140]."Process Value";
   "Unit1.MotionNodes".PLCToMotion.Parameters.StackMain.StackCalculate.Time.PnPZUpStart := "HMI_Interface_Parameter".Parameter_Text[141]."Process Value";
   "Unit1.MotionNodes".PLCToMotion.Parameters.StackMain.StackCalculate.Time.PnPZUpEnd := "HMI_Interface_Parameter".Parameter_Text[142]."Process Value";
   "Unit1.MotionNodes".PLCToMotion.Parameters.StackMain.StackCalculate.Time.MandrelBwdStart := "HMI_Interface_Parameter".Parameter_Text[143]."Process Value";
   "Unit1.MotionNodes".PLCToMotion.Parameters.StackMain.StackCalculate.Time.MandrelBwdEnd := "HMI_Interface_Parameter".Parameter_Text[144]."Process Value";
   "Unit1.MotionNodes".PLCToMotion.Parameters.StackMain.StackCalculate.Time.MandrelFwdStart := "HMI_Interface_Parameter".Parameter_Text[145]."Process Value";
   "Unit1.MotionNodes".PLCToMotion.Parameters.StackMain.StackCalculate.Time.MandrelFwdEnd := "HMI_Interface_Parameter".Parameter_Text[146]."Process Value";
   "Unit1.MotionNodes".PLCToMotion.Parameters.StackMain.StackCalculate.Time.MandrelUpStart1 := "HMI_Interface_Parameter".Parameter_Text[147]."Process Value";
   "Unit1.MotionNodes".PLCToMotion.Parameters.StackMain.StackCalculate.Time.MandrelUpEnd1 := "HMI_Interface_Parameter".Parameter_Text[148]."Process Value";
   "Unit1.MotionNodes".PLCToMotion.Parameters.StackMain.StackCalculate.Time.MandrelUpStart2 := "HMI_Interface_Parameter".Parameter_Text[149]."Process Value";
   "Unit1.MotionNodes".PLCToMotion.Parameters.StackMain.StackCalculate.Time.MandrelUpEnd2 := "HMI_Interface_Parameter".Parameter_Text[150]."Process Value";
   "Unit1.MotionNodes".PLCToMotion.Parameters.StackMain.StackCalculate.Time.MandrelDownStart := "HMI_Interface_Parameter".Parameter_Text[151]."Process Value";
   "Unit1.MotionNodes".PLCToMotion.Parameters.StackMain.StackCalculate.Time.MandrelDownEnd := "HMI_Interface_Parameter".Parameter_Text[152]."Process Value";
   "Unit1.MotionNodes".PLCToMotion.Parameters.StackMain.StackCalculate.Position.FinalRollerBwdPos := "HMI_Interface_Parameter".Parameter_Text[153]."Process Value";
   "Unit1.MotionNodes".PLCToMotion.Parameters.StackMain.StackCalculate.Position.FinalRollerFwdPos := "HMI_Interface_Parameter".Parameter_Text[154]."Process Value";
END_REGION

REGION Network 6 (SCL): HMI Parameter Image Process Value
   // Move to recipe (Network 7)
   //"HMI_Interface_Parameter".Parameter_Image[0]."Process Value" := Unit1.Em3.HmiInterface.auxiliary.dancerRegulator;
   //"HMI_Interface_Parameter".Parameter_Image[1]."Process Value" := Unit1.Em0.HmiInterface.auxiliary.AutoSpliceRemainingLength;
   //
   //"HMI_Interface_Parameter".Parameter_Image[1]."Process Value" := Unit1.Em1.HmiInterface.auxiliary.AutoSpliceRemainingLength;
END_REGION

REGION Network 7 (SCL): PLC -> Motion Teaching Start / End Pos (YS)
   /// Start Pos
   //
   "Unit1.MotionNodes".PLCToMotion.Parameters.StackMain.StackCalculate.TeachingPos.StartPos.Compensator := "Unit1.Em3.Config".cmCompensatorAxisX.setPositions[0].position;
   "Unit1.MotionNodes".PLCToMotion.Parameters.StackMain.StackCalculate.TeachingPos.StartPos.FinalRoller := "Unit1.Em6.Config".cmFinalRollerFrontAxisX.setPositions[0].position;

   "Unit1.MotionNodes".PLCToMotion.Parameters.StackMain.StackCalculate.TeachingPos.StartPos.AnodePnPX1 := "Unit1.Em4.Config".cmAnodeMainPnP1AxisX.setPositions[0].position;
   "Unit1.MotionNodes".PLCToMotion.Parameters.StackMain.StackCalculate.TeachingPos.StartPos.AnodePnPX2 := "Unit1.Em4.Config".cmAnodeMainPnP2AxisX.setPositions[0].position;
   "Unit1.MotionNodes".PLCToMotion.Parameters.StackMain.StackCalculate.TeachingPos.StartPos.AnodePnPZ1 := "Unit1.Em4.Config".cmAnodeMainPnP1AxisZ.setPositions[0].position;
   "Unit1.MotionNodes".PLCToMotion.Parameters.StackMain.StackCalculate.TeachingPos.StartPos.AnodePnPZ2 := "Unit1.Em4.Config".cmAnodeMainPnP2AxisZ.setPositions[0].position;

   "Unit1.MotionNodes".PLCToMotion.Parameters.StackMain.StackCalculate.TeachingPos.StartPos.CathodePnPX1 := "Unit1.Em5.Config".cmCathodeMainPnP1AxisX.setPositions[0].position;
   "Unit1.MotionNodes".PLCToMotion.Parameters.StackMain.StackCalculate.TeachingPos.StartPos.CathodePnPX2 := "Unit1.Em5.Config".cmCathodeMainPnP2AxisX.setPositions[0].position;
   "Unit1.MotionNodes".PLCToMotion.Parameters.StackMain.StackCalculate.TeachingPos.StartPos.CathodePnPZ1 := "Unit1.Em5.Config".cmCathodeMainPnP1AxisZ.setPositions[0].position;
   "Unit1.MotionNodes".PLCToMotion.Parameters.StackMain.StackCalculate.TeachingPos.StartPos.CathodePnPZ2 := "Unit1.Em5.Config".cmCathodeMainPnP2AxisZ.setPositions[0].position;

   "Unit1.MotionNodes".PLCToMotion.Parameters.StackMain.StackCalculate.TeachingPos.StartPos.AnodeMandrelYFront := "Unit1.Em6.Config".cmMendrelAnodeFrontAxisY.setPositions[0].position;
   "Unit1.MotionNodes".PLCToMotion.Parameters.StackMain.StackCalculate.TeachingPos.StartPos.AnodeMandrelYRear := "Unit1.Em6.Config".cmMendrelAnodeRearAxisY.setPositions[0].position;
   "Unit1.MotionNodes".PLCToMotion.Parameters.StackMain.StackCalculate.TeachingPos.StartPos.AnodeMandrelZFront := "Unit1.Em6.Config".cmMendrelAnodeFrontAxisZ.setPositions[0].position;
   "Unit1.MotionNodes".PLCToMotion.Parameters.StackMain.StackCalculate.TeachingPos.StartPos.AnodeMandrelZRear := "Unit1.Em6.Config".cmMendrelAnodeRearAxisZ.setPositions[0].position;
   "Unit1.MotionNodes".PLCToMotion.Parameters.StackMain.StackCalculate.TeachingPos.StartPos.CathodeMandrelYFront := "Unit1.Em6.Config".cmMendrelCathodeFrontAxisY.setPositions[0].position;
   "Unit1.MotionNodes".PLCToMotion.Parameters.StackMain.StackCalculate.TeachingPos.StartPos.CathodeMandrelYRear := "Unit1.Em6.Config".cmMendrelCathodeRearAxisY.setPositions[0].position;
   "Unit1.MotionNodes".PLCToMotion.Parameters.StackMain.StackCalculate.TeachingPos.StartPos.CathodeMandrelZFront := "Unit1.Em6.Config".cmMendrelCathodeFrontAxisZ.setPositions[0].position;
   "Unit1.MotionNodes".PLCToMotion.Parameters.StackMain.StackCalculate.TeachingPos.StartPos.CathodeMandrelZRear := "Unit1.Em6.Config".cmMendrelCathodeRearAxisZ.setPositions[0].position;

   ///// End Pos

   "Unit1.MotionNodes".PLCToMotion.Parameters.StackMain.StackCalculate.TeachingPos.EndPos.FinalRoller := "Unit1.Em6.Config".cmFinalRollerFrontAxisX.setPositions[1].position;
   "Unit1.MotionNodes".PLCToMotion.Parameters.StackMain.StackCalculate.TeachingPos.EndPos.AnodePnPX1 := "Unit1.Em4.Config".cmAnodeMainPnP1AxisX.setPositions[1].position;
   "Unit1.MotionNodes".PLCToMotion.Parameters.StackMain.StackCalculate.TeachingPos.EndPos.AnodePnPX2 := "Unit1.Em4.Config".cmAnodeMainPnP2AxisX.setPositions[1].position;

   "Unit1.MotionNodes".PLCToMotion.Parameters.StackMain.StackCalculate.TeachingPos.EndPos.AnodePnPZ1P1 := "Unit1.Em4.Config".cmAnodeMainPnP1AxisZ.setPositions[1].position;
   "Unit1.MotionNodes".PLCToMotion.Parameters.StackMain.StackCalculate.TeachingPos.EndPos.AnodePnPZ1P2 := "Unit1.Em4.Config".cmAnodeMainPnP1AxisZ.setPositions[2].position;
   "Unit1.MotionNodes".PLCToMotion.Parameters.StackMain.StackCalculate.TeachingPos.EndPos.AnodePnPZ2P1 := "Unit1.Em4.Config".cmAnodeMainPnP2AxisZ.setPositions[1].position;
   "Unit1.MotionNodes".PLCToMotion.Parameters.StackMain.StackCalculate.TeachingPos.EndPos.AnodePnPZ2P2 := "Unit1.Em4.Config".cmAnodeMainPnP2AxisZ.setPositions[2].position;

   "Unit1.MotionNodes".PLCToMotion.Parameters.StackMain.StackCalculate.TeachingPos.EndPos.CathodePnPX1 := "Unit1.Em5.Config".cmCathodeMainPnP1AxisX.setPositions[1].position;
   "Unit1.MotionNodes".PLCToMotion.Parameters.StackMain.StackCalculate.TeachingPos.EndPos.CathodePnPX2 := "Unit1.Em5.Config".cmCathodeMainPnP2AxisX.setPositions[1].position;

   "Unit1.MotionNodes".PLCToMotion.Parameters.StackMain.StackCalculate.TeachingPos.EndPos.CathodePnPZ1P1 := "Unit1.Em5.Config".cmCathodeMainPnP1AxisZ.setPositions[1].position;
   "Unit1.MotionNodes".PLCToMotion.Parameters.StackMain.StackCalculate.TeachingPos.EndPos.CathodePnPZ1P2 := "Unit1.Em5.Config".cmCathodeMainPnP1AxisZ.setPositions[2].position;
   "Unit1.MotionNodes".PLCToMotion.Parameters.StackMain.StackCalculate.TeachingPos.EndPos.CathodePnPZ2P1 := "Unit1.Em5.Config".cmCathodeMainPnP2AxisZ.setPositions[1].position;
   "Unit1.MotionNodes".PLCToMotion.Parameters.StackMain.StackCalculate.TeachingPos.EndPos.CathodePnPZ2P2 := "Unit1.Em5.Config".cmCathodeMainPnP2AxisZ.setPositions[2].position;


   "Unit1.MotionNodes".PLCToMotion.Parameters.StackMain.StackCalculate.TeachingPos.EndPos.AnodeMandrelYFront := "Unit1.Em6.Config".cmMendrelAnodeFrontAxisY.setPositions[1].position;
   "Unit1.MotionNodes".PLCToMotion.Parameters.StackMain.StackCalculate.TeachingPos.EndPos.AnodeMandrelYRear := "Unit1.Em6.Config".cmMendrelAnodeRearAxisY.setPositions[1].position;
   "Unit1.MotionNodes".PLCToMotion.Parameters.StackMain.StackCalculate.TeachingPos.EndPos.AnodeMandrelZFront := "Unit1.Em6.Config".cmMendrelAnodeFrontAxisZ.setPositions[1].position;
   "Unit1.MotionNodes".PLCToMotion.Parameters.StackMain.StackCalculate.TeachingPos.EndPos.AnodeMandrelZRear := "Unit1.Em6.Config".cmMendrelAnodeRearAxisZ.setPositions[1].position;
   "Unit1.MotionNodes".PLCToMotion.Parameters.StackMain.StackCalculate.TeachingPos.EndPos.CathodeMandrelYFront := "Unit1.Em6.Config".cmMendrelCathodeFrontAxisY.setPositions[1].position;
   "Unit1.MotionNodes".PLCToMotion.Parameters.StackMain.StackCalculate.TeachingPos.EndPos.CathodeMandrelYRear := "Unit1.Em6.Config".cmMendrelCathodeRearAxisY.setPositions[1].position;
   "Unit1.MotionNodes".PLCToMotion.Parameters.StackMain.StackCalculate.TeachingPos.EndPos.CathodeMandrelZFront := "Unit1.Em6.Config".cmMendrelCathodeFrontAxisZ.setPositions[1].position;
   "Unit1.MotionNodes".PLCToMotion.Parameters.StackMain.StackCalculate.TeachingPos.EndPos.CathodeMandrelZRear := "Unit1.Em6.Config".cmMendrelCathodeRearAxisZ.setPositions[1].position;
END_REGION

REGION Network 8 (SCL): PLC -> HMI Softcam
   "HMI_Interface_Parameter".Softcam[1] := "Unit1.Em0.HmiInterface".cm.softCam.unwinderTopAxisB;
   "HMI_Interface_Parameter".Softcam[2] := "Unit1.Em1.HmiInterface".cm.softCam.unwinderBtmAxisB;
   "HMI_Interface_Parameter".Softcam[3] := "Unit1.Em3.HmiInterface".cm.softCam.compensatorAxisX;
   "HMI_Interface_Parameter".Softcam[4] := "Unit1.Em7.HmiInterface".cm.softCam.jrPusherAxisZ;
   "HMI_Interface_Parameter".Softcam[5] := "Unit1.Em4.HmiInterface".cm.softCam.anodeMainPnP1AxisX;
   "HMI_Interface_Parameter".Softcam[6] := "Unit1.Em4.HmiInterface".cm.softCam.anodeMainPnP2AxisX;
   "HMI_Interface_Parameter".Softcam[7] := "Unit1.Em5.HmiInterface".cm.softCam.cathodeMainPnP1AxisX;
   "HMI_Interface_Parameter".Softcam[8] := "Unit1.Em5.HmiInterface".cm.softCam.cathodeMainPnP2AxisX;
   "HMI_Interface_Parameter".Softcam[9] := "Unit1.Em5.HmiInterface".cm.softCam.cathodeMainPnP1AxisY;
   "HMI_Interface_Parameter".Softcam[10] := "Unit1.Em5.HmiInterface".cm.softCam.cathodeMainPnP1AxisZ;
   "HMI_Interface_Parameter".Softcam[11] := "Unit1.Em4.HmiInterface".cm.softCam.anodeMainPnP1AxisY;
   "HMI_Interface_Parameter".Softcam[12] := "Unit1.Em4.HmiInterface".cm.softCam.anodeMainPnP1AxisZ;
   "HMI_Interface_Parameter".Softcam[13] := "Unit1.Em5.HmiInterface".cm.softCam.cathodeMainPnP2AxisZ;
   "HMI_Interface_Parameter".Softcam[14] := "Unit1.Em4.HmiInterface".cm.softCam.anodeMainPnP2AxisZ;
   "HMI_Interface_Parameter".Softcam[15] := "Unit1.Em4.HmiInterface".cm.softCam.anodeAlignTableAxisX;
   "HMI_Interface_Parameter".Softcam[16] := "Unit1.Em4.HmiInterface".cm.softCam.anodeAlignTableAxisY2;
   "HMI_Interface_Parameter".Softcam[17] := "Unit1.Em4.HmiInterface".cm.softCam.anodeAlignTableAxisY1;
   "HMI_Interface_Parameter".Softcam[18] := "Unit1.Em5.HmiInterface".cm.softCam.cathodeAlignTableAxisX;
   "HMI_Interface_Parameter".Softcam[19] := "Unit1.Em5.HmiInterface".cm.softCam.cathodeAlignTableAxisY2;
   "HMI_Interface_Parameter".Softcam[20] := "Unit1.Em5.HmiInterface".cm.softCam.cathodeAlignTableAxisY1;
   "HMI_Interface_Parameter".Softcam[21] := "Unit1.Em6.HmiInterface".cm.softCam.finalRollerFrontAxisX;
   "HMI_Interface_Parameter".Softcam[22] := "Unit1.Em6.HmiInterface".cm.softCam.finalRollerRearAxisX;
   "HMI_Interface_Parameter".Softcam[23] := "Unit1.Em6.HmiInterface".cm.softCam.mendrelAnodeFrontAxisY;
   "HMI_Interface_Parameter".Softcam[24] := "Unit1.Em6.HmiInterface".cm.softCam.mendrelAnodeFrontAxisZ;
   "HMI_Interface_Parameter".Softcam[25] := "Unit1.Em6.HmiInterface".cm.softCam.mendrelAnodeRearAxisY;
   "HMI_Interface_Parameter".Softcam[26] := "Unit1.Em6.HmiInterface".cm.softCam.mendrelAnodeRearAxisZ;
   "HMI_Interface_Parameter".Softcam[27] := "Unit1.Em6.HmiInterface".cm.softCam.mendrelCathodeFrontAxisY;
   "HMI_Interface_Parameter".Softcam[28] := "Unit1.Em6.HmiInterface".cm.softCam.mendrelCathodeFrontAxisZ;
   "HMI_Interface_Parameter".Softcam[29] := "Unit1.Em6.HmiInterface".cm.softCam.mendrelCathodeRearAxisY;
   "HMI_Interface_Parameter".Softcam[30] := "Unit1.Em6.HmiInterface".cm.softCam.mendrelCathodeRearAxisZ;
   "HMI_Interface_Parameter".Softcam[31] := "Unit1.Em6.HmiInterface".cm.softCam.stackTableAxisZ;
   "HMI_Interface_Parameter".Softcam[32] := "Unit1.Em6.HmiInterface".cm.softCam.stackTableOutFrontAxisZ;
   "HMI_Interface_Parameter".Softcam[33] := "Unit1.Em6.HmiInterface".cm.softCam.stackTableOutRearAxisZ;
   "HMI_Interface_Parameter".Softcam[34] := "Unit1.Em7.HmiInterface".cm.softCam.sepaClampnCutterAxisX;
   "HMI_Interface_Parameter".Softcam[35] := "Unit1.Em7.HmiInterface".cm.softCam.sepaClampnCutterAxisZ;
   "HMI_Interface_Parameter".Softcam[36] := "Unit1.Em7.HmiInterface".cm.softCam.sepaGripperAxisX;
   "HMI_Interface_Parameter".Softcam[37] := "Unit1.Em7.HmiInterface".cm.softCam.sepaGripperAxisZ;
   "HMI_Interface_Parameter".Softcam[38] := "Unit1.Em7.HmiInterface".cm.softCam.sepaGripperAxisC;
   "HMI_Interface_Parameter".Softcam[39] := "Unit1.Em7.HmiInterface".cm.softCam.jrWinderRearAxisY;
   "HMI_Interface_Parameter".Softcam[40] := "Unit1.Em7.HmiInterface".cm.softCam.jrWinderFrontAxisY;
   "HMI_Interface_Parameter".Softcam[41] := "Unit1.Em7.HmiInterface".cm.softCam.jrWinderAxisB;
END_REGION

REGION Network 9 (SCL): SamplingMode Complete end
   IF "Unit1.EmNodes".SamplingModeComplete THEN
       "HMI_Interface_Parameter".FATModeInterface.ModeSelect.SamplingMode := FALSE;
       ;
   END_IF;
END_REGION

REGION Network 10: SamplingMode Btn on count reset trigger // cell current count
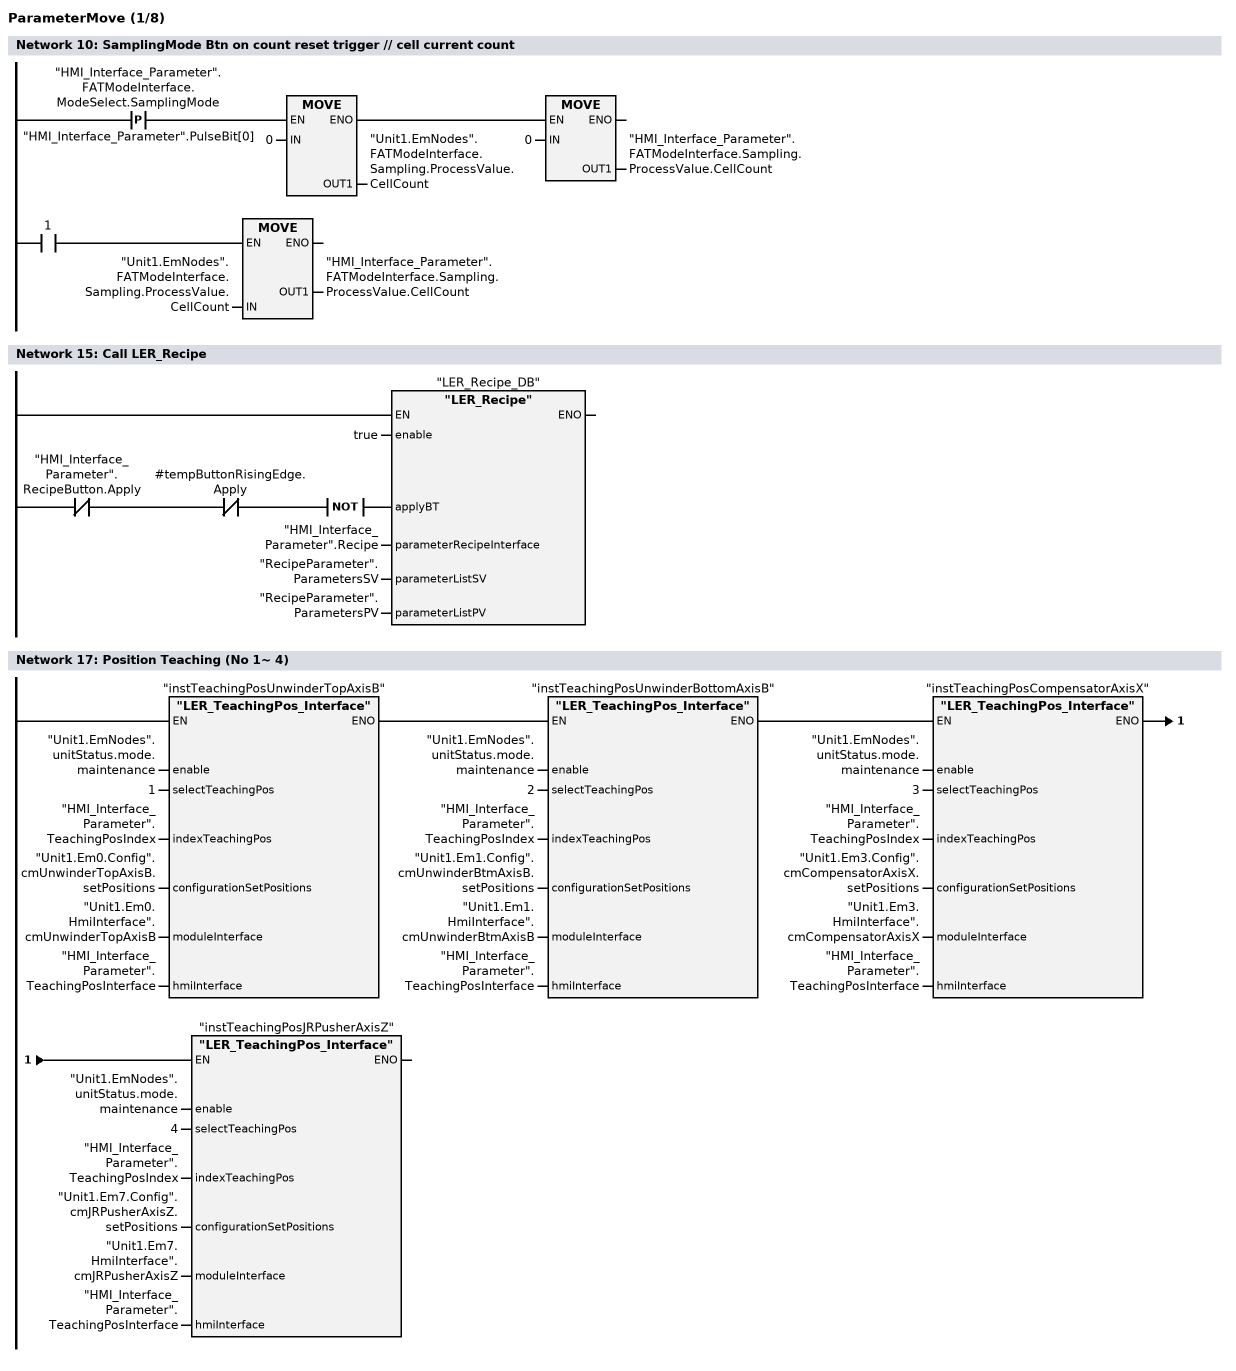
   RUNG wire#powerrail
      P_Contact(operand := "HMI_Interface_Parameter".FATModeInterface.ModeSelect.SamplingMode, bit := "HMI_Interface_Parameter".PulseBit[0])
      Move(in := 0, out1 => "Unit1.EmNodes".FATModeInterface.Sampling.ProcessValue.CellCount)
      Move(in := 0, out1 => "HMI_Interface_Parameter".FATModeInterface.Sampling.ProcessValue.CellCount)
   END_RUNG
   RUNG wire#powerrail
      Contact( 1 )
      Move(in := "Unit1.EmNodes".FATModeInterface.Sampling.ProcessValue.CellCount, out1 => "HMI_Interface_Parameter".FATModeInterface.Sampling.ProcessValue.CellCount)
   END_RUNG
   // the same network as SCL:
   #_w1 := "HMI_Interface_Parameter".FATModeInterface.ModeSelect.SamplingMode AND NOT "HMI_Interface_Parameter".PulseBit[0];   // rising edge of "HMI_Interface_Parameter".FATModeInterface.ModeSelect.SamplingMode
   "HMI_Interface_Parameter".PulseBit[0] := "HMI_Interface_Parameter".FATModeInterface.ModeSelect.SamplingMode;
   IF #_w1 THEN
       "Unit1.EmNodes".FATModeInterface.Sampling.ProcessValue.CellCount := 0;
       "HMI_Interface_Parameter".FATModeInterface.Sampling.ProcessValue.CellCount := 0;
   END_IF;
   IF 1 THEN
       "HMI_Interface_Parameter".FATModeInterface.Sampling.ProcessValue.CellCount := "Unit1.EmNodes".FATModeInterface.Sampling.ProcessValue.CellCount;
   END_IF;
END_REGION

REGION Network 12 (SCL): HMI Interface Parameter To Recipe Pareameter SV
   // IF #tempButtonRisingEdge.Apply THEN
   //     "RecipeParameter".ParametersSV.Recipe1 := "HMI_Interface_Parameter"."Default Recipe".SetValue."Electrode Width".Anode;
   //     "RecipeParameter".ParametersSV.Recipe2 := "HMI_Interface_Parameter"."Default Recipe".SetValue."Electrode Width".Cathode;
   //     "RecipeParameter".ParametersSV.Recipe3 := "HMI_Interface_Parameter"."Default Recipe".SetValue."Anode Thinkness";
   //     "RecipeParameter".ParametersSV.Recipe4 := "HMI_Interface_Parameter"."Default Recipe".SetValue."Cathode Thinkness";
   //     "RecipeParameter".ParametersSV.Recipe5 := "HMI_Interface_Parameter"."Default Recipe".SetValue."Sperator Thinkness";
   //     "RecipeParameter".ParametersSV.Recipe6 := "HMI_Interface_Parameter"."Default Recipe".SetValue."Jelly Roll Width";
   //     "RecipeParameter".ParametersSV.Recipe7 := "HMI_Interface_Parameter"."Default Recipe".SetValue."Cell Stack Count";
   //     "RecipeParameter".ParametersSV.Recipe8 := "HMI_Interface_Parameter".Parameter_Image[0]."Set Value";
   //     "RecipeParameter".ParametersSV.Recipe9 := "HMI_Interface_Parameter".Parameter_Image[1]."Set Value";
   //     //
   //     //"RecipeParameter".ParametersSV.Recipe10 := ;
   //     //"RecipeParameter".ParametersSV.Recipe11 := ;
   //     //"RecipeParameter".ParametersSV.Recipe12 := ;
   //     //"RecipeParameter".ParametersSV.Recipe13 := ;
   //     //"RecipeParameter".ParametersSV.Recipe14 := ;
   //     //"RecipeParameter".ParametersSV.Recipe15 := ;
   //     //"RecipeParameter".ParametersSV.Recipe16 := ;
   //     //"RecipeParameter".ParametersSV.Recipe17 := ;
   //     //"RecipeParameter".ParametersSV.Recipe18 := ;
   //     //"RecipeParameter".ParametersSV.Recipe19 := ;
   //     //"RecipeParameter".ParametersSV.Recipe20 := ;
   //     //"RecipeParameter".ParametersSV.Recipe21 := ;
   //     //"RecipeParameter".ParametersSV.Recipe22 := ;
   //     //"RecipeParameter".ParametersSV.Recipe23 := ;
   //     //"RecipeParameter".ParametersSV.Recipe24 := ;
   //     //"RecipeParameter".ParametersSV.Recipe25 := ;
   // END_IF;
END_REGION

REGION Network 13 (SCL): HMI Interface Pareameter Recipe Data To HMI Interface Parameter Process Value
   // IF "HMI_Interface_Parameter".Recipe.RecipeChangeBT OR "HMI_Interface_Parameter".RecipeButton.Apply OR #tempButtonRisingEdge.Apply THEN

   //     "HMI_Interface_Parameter"."Default Recipe".ProcessValue."Electrode Width".Anode := "HMI_Interface_Parameter".Recipe.Recipe_Data["HMI_Interface_Parameter".Recipe.CurrentRecipeNum].Recipe1;
   //     "HMI_Interface_Parameter"."Default Recipe".ProcessValue."Electrode Width".Cathode := "HMI_Interface_Parameter".Recipe.Recipe_Data["HMI_Interface_Parameter".Recipe.CurrentRecipeNum].Recipe2;
   //     "HMI_Interface_Parameter"."Default Recipe".ProcessValue."Anode Thinkness" := "HMI_Interface_Parameter".Recipe.Recipe_Data["HMI_Interface_Parameter".Recipe.CurrentRecipeNum].Recipe3;
   //     "HMI_Interface_Parameter"."Default Recipe".ProcessValue."Cathode Thinkness" := "HMI_Interface_Parameter".Recipe.Recipe_Data["HMI_Interface_Parameter".Recipe.CurrentRecipeNum].Recipe4;
   //     "HMI_Interface_Parameter"."Default Recipe".ProcessValue."Sperator Thinkness" := "HMI_Interface_Parameter".Recipe.Recipe_Data["HMI_Interface_Parameter".Recipe.CurrentRecipeNum].Recipe5;
   //     "HMI_Interface_Parameter"."Default Recipe".ProcessValue."Jelly Roll Width" := "HMI_Interface_Parameter".Recipe.Recipe_Data["HMI_Interface_Parameter".Recipe.CurrentRecipeNum].Recipe6;
   //     "HMI_Interface_Parameter"."Default Recipe".ProcessValue."Cell Stack Count" := LREAL_TO_SINT("HMI_Interface_Parameter".Recipe.Recipe_Data["HMI_Interface_Parameter".Recipe.CurrentRecipeNum].Recipe7);
   //     "HMI_Interface_Parameter".Parameter_Image[0]."Process Value" := "HMI_Interface_Parameter".Recipe.Recipe_Data["HMI_Interface_Parameter".Recipe.CurrentRecipeNum].Recipe8;
   //     "HMI_Interface_Parameter".Parameter_Image[1]."Process Value" := "HMI_Interface_Parameter".Recipe.Recipe_Data["HMI_Interface_Parameter".Recipe.CurrentRecipeNum].Recipe9;
   //     // := "HMI_Interface_Parameter".Recipe.Recipe_Data["HMI_Interface_Parameter".Recipe.CurrentRecipeNum].Recipe10;
   //     // := "HMI_Interface_Parameter".Recipe.Recipe_Data["HMI_Interface_Parameter".Recipe.CurrentRecipeNum].Recipe11;
   //     // := "HMI_Interface_Parameter".Recipe.Recipe_Data["HMI_Interface_Parameter".Recipe.CurrentRecipeNum].Recipe12;
   //     // := "HMI_Interface_Parameter".Recipe.Recipe_Data["HMI_Interface_Parameter".Recipe.CurrentRecipeNum].Recipe13;
   //     // := "HMI_Interface_Parameter".Recipe.Recipe_Data["HMI_Interface_Parameter".Recipe.CurrentRecipeNum].Recipe14;
   //     // := "HMI_Interface_Parameter".Recipe.Recipe_Data["HMI_Interface_Parameter".Recipe.CurrentRecipeNum].Recipe15;
   // END_IF;
END_REGION

REGION Network 14 (SCL): Recipe Parameter PV To Unit EmData Recipe
   "Unit1.EmData".UnitRecipe.size.Anode.length := "RecipeParameter".ParametersPV.Recipe1;
   "Unit1.EmData".UnitRecipe.size.Cathode.length := "RecipeParameter".ParametersPV.Recipe2;
   "Unit1.EmData".UnitRecipe.size.Anode.thickness := "RecipeParameter".ParametersPV.Recipe3;
   "Unit1.EmData".UnitRecipe.size.Cathode.thickness := "RecipeParameter".ParametersPV.Recipe4;
   "Unit1.EmData".UnitRecipe.SepaThickness := "RecipeParameter".ParametersPV.Recipe5;
   "Unit1.EmData".UnitRecipe.JellyRollWidth := "RecipeParameter".ParametersPV.Recipe6;
   "Unit1.EmData".UnitRecipe.StackCount := "RecipeParameter".ParametersPV.Recipe7;
   "Unit1.EmData".UnitRecipe.DancerRegulator := "RecipeParameter".ParametersPV.Recipe8;
   "Unit1.EmData".UnitRecipe.AutoSpliceRemainingLength := "RecipeParameter".ParametersPV.Recipe9;
   //
   // := "RecipeParameter".ParametersPV.Recipe10;
   // := "RecipeParameter".ParametersPV.Recipe11;
   // := "RecipeParameter".ParametersPV.Recipe12;
   // := "RecipeParameter".ParametersPV.Recipe13;
   // := "RecipeParameter".ParametersPV.Recipe14;
   // := "RecipeParameter".ParametersPV.Recipe15;
END_REGION

REGION Network 15: Call LER_Recipe
   RUNG wire#powerrail
      "LER_Recipe_DB"(applyBT := wire#w1, enable := true, parameterRecipeInterface := "HMI_Interface_Parameter".Recipe, parameterListSV := "RecipeParameter".ParametersSV, parameterListPV := "RecipeParameter".ParametersPV)
   END_RUNG
   RUNG wire#powerrail
      I_Contact( "HMI_Interface_Parameter".RecipeButton.Apply )
      I_Contact( #tempButtonRisingEdge.Apply )
      Not()
   END_RUNG wire#w1
   // the same network as SCL:
   "LER_Recipe_DB"(enable := true,   // "LER_Recipe"
                   applyBT := NOT (NOT "HMI_Interface_Parameter".RecipeButton.Apply AND NOT #tempButtonRisingEdge.Apply),
                   parameterRecipeInterface := "HMI_Interface_Parameter".Recipe,
                   parameterListSV := "RecipeParameter".ParametersSV,
                   parameterListPV := "RecipeParameter".ParametersPV);
END_REGION

REGION Network 17: Position Teaching (No 1~ 4)
   RUNG wire#powerrail
      "instTeachingPosUnwinderTopAxisB"(enable := "Unit1.EmNodes".unitStatus.mode.maintenance, selectTeachingPos := 1, indexTeachingPos := "HMI_Interface_Parameter".TeachingPosIndex, configurationSetPositions := "Unit1.Em0.Config".cmUnwinderTopAxisB.setPositions, moduleInterface := "Unit1.Em0.HmiInterface".cmUnwinderTopAxisB, hmiInterface := "HMI_Interface_Parameter".TeachingPosInterface)
      "instTeachingPosUnwinderBottomAxisB"(enable := "Unit1.EmNodes".unitStatus.mode.maintenance, selectTeachingPos := 2, indexTeachingPos := "HMI_Interface_Parameter".TeachingPosIndex, configurationSetPositions := "Unit1.Em1.Config".cmUnwinderBtmAxisB.setPositions, moduleInterface := "Unit1.Em1.HmiInterface".cmUnwinderBtmAxisB, hmiInterface := "HMI_Interface_Parameter".TeachingPosInterface)
      "instTeachingPosCompensatorAxisX"(enable := "Unit1.EmNodes".unitStatus.mode.maintenance, selectTeachingPos := 3, indexTeachingPos := "HMI_Interface_Parameter".TeachingPosIndex, configurationSetPositions := "Unit1.Em3.Config".cmCompensatorAxisX.setPositions, moduleInterface := "Unit1.Em3.HmiInterface".cmCompensatorAxisX, hmiInterface := "HMI_Interface_Parameter".TeachingPosInterface)
      "instTeachingPosJRPusherAxisZ"(enable := "Unit1.EmNodes".unitStatus.mode.maintenance, selectTeachingPos := 4, indexTeachingPos := "HMI_Interface_Parameter".TeachingPosIndex, configurationSetPositions := "Unit1.Em7.Config".cmJRPusherAxisZ.setPositions, moduleInterface := "Unit1.Em7.HmiInterface".cmJRPusherAxisZ, hmiInterface := "HMI_Interface_Parameter".TeachingPosInterface)
   END_RUNG
   // the same network as SCL:
   "instTeachingPosUnwinderTopAxisB"(enable := "Unit1.EmNodes".unitStatus.mode.maintenance,   // "LER_TeachingPos_Interface"
                           selectTeachingPos := 1,
                           indexTeachingPos := "HMI_Interface_Parameter".TeachingPosIndex,
                           configurationSetPositions := "Unit1.Em0.Config".cmUnwinderTopAxisB.setPositions,
                           moduleInterface := "Unit1.Em0.HmiInterface".cmUnwinderTopAxisB,
                           hmiInterface := "HMI_Interface_Parameter".TeachingPosInterface,
                           ENO => #_w1);
   "instTeachingPosUnwinderBottomAxisB"(EN := #_w1,   // "LER_TeachingPos_Interface"
                           enable := "Unit1.EmNodes".unitStatus.mode.maintenance,
                           selectTeachingPos := 2,
                           indexTeachingPos := "HMI_Interface_Parameter".TeachingPosIndex,
                           configurationSetPositions := "Unit1.Em1.Config".cmUnwinderBtmAxisB.setPositions,
                           moduleInterface := "Unit1.Em1.HmiInterface".cmUnwinderBtmAxisB,
                           hmiInterface := "HMI_Interface_Parameter".TeachingPosInterface,
                           ENO => #_w2);
   "instTeachingPosCompensatorAxisX"(EN := #_w2,   // "LER_TeachingPos_Interface"
                           enable := "Unit1.EmNodes".unitStatus.mode.maintenance,
                           selectTeachingPos := 3,
                           indexTeachingPos := "HMI_Interface_Parameter".TeachingPosIndex,
                           configurationSetPositions := "Unit1.Em3.Config".cmCompensatorAxisX.setPositions,
                           moduleInterface := "Unit1.Em3.HmiInterface".cmCompensatorAxisX,
                           hmiInterface := "HMI_Interface_Parameter".TeachingPosInterface,
                           ENO => #_w3);
   IF #_w3 THEN
       "instTeachingPosJRPusherAxisZ"(enable := "Unit1.EmNodes".unitStatus.mode.maintenance,   // "LER_TeachingPos_Interface"
                               selectTeachingPos := 4,
                               indexTeachingPos := "HMI_Interface_Parameter".TeachingPosIndex,
                               configurationSetPositions := "Unit1.Em7.Config".cmJRPusherAxisZ.setPositions,
                               moduleInterface := "Unit1.Em7.HmiInterface".cmJRPusherAxisZ,
                               hmiInterface := "HMI_Interface_Parameter".TeachingPosInterface);
   END_IF;
END_REGION

REGION Network 18: Position Teaching (No 5~8)
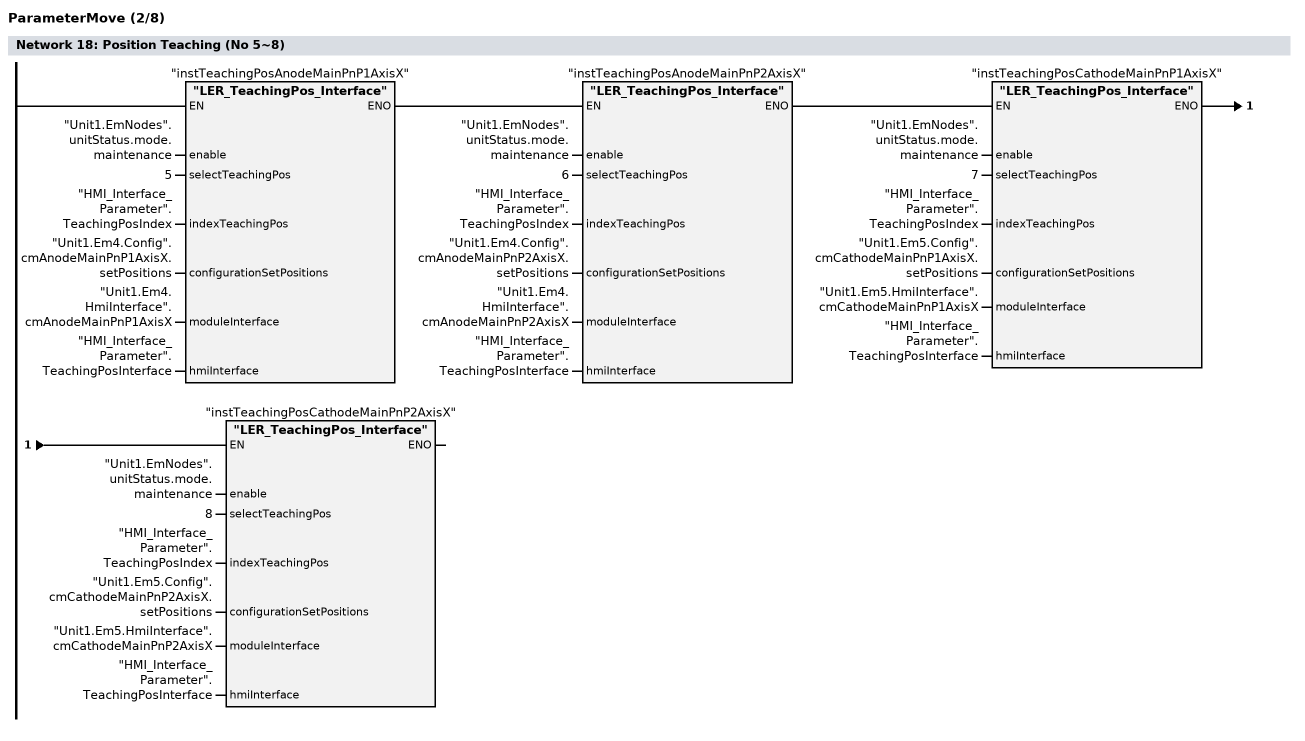
   RUNG wire#powerrail
      "instTeachingPosAnodeMainPnP1AxisX"(enable := "Unit1.EmNodes".unitStatus.mode.maintenance, selectTeachingPos := 5, indexTeachingPos := "HMI_Interface_Parameter".TeachingPosIndex, configurationSetPositions := "Unit1.Em4.Config".cmAnodeMainPnP1AxisX.setPositions, moduleInterface := "Unit1.Em4.HmiInterface".cmAnodeMainPnP1AxisX, hmiInterface := "HMI_Interface_Parameter".TeachingPosInterface)
      "instTeachingPosAnodeMainPnP2AxisX"(enable := "Unit1.EmNodes".unitStatus.mode.maintenance, selectTeachingPos := 6, indexTeachingPos := "HMI_Interface_Parameter".TeachingPosIndex, configurationSetPositions := "Unit1.Em4.Config".cmAnodeMainPnP2AxisX.setPositions, moduleInterface := "Unit1.Em4.HmiInterface".cmAnodeMainPnP2AxisX, hmiInterface := "HMI_Interface_Parameter".TeachingPosInterface)
      "instTeachingPosCathodeMainPnP1AxisX"(enable := "Unit1.EmNodes".unitStatus.mode.maintenance, selectTeachingPos := 7, indexTeachingPos := "HMI_Interface_Parameter".TeachingPosIndex, configurationSetPositions := "Unit1.Em5.Config".cmCathodeMainPnP1AxisX.setPositions, moduleInterface := "Unit1.Em5.HmiInterface".cmCathodeMainPnP1AxisX, hmiInterface := "HMI_Interface_Parameter".TeachingPosInterface)
      "instTeachingPosCathodeMainPnP2AxisX"(enable := "Unit1.EmNodes".unitStatus.mode.maintenance, selectTeachingPos := 8, indexTeachingPos := "HMI_Interface_Parameter".TeachingPosIndex, configurationSetPositions := "Unit1.Em5.Config".cmCathodeMainPnP2AxisX.setPositions, moduleInterface := "Unit1.Em5.HmiInterface".cmCathodeMainPnP2AxisX, hmiInterface := "HMI_Interface_Parameter".TeachingPosInterface)
   END_RUNG
   // the same network as SCL:
   "instTeachingPosAnodeMainPnP1AxisX"(enable := "Unit1.EmNodes".unitStatus.mode.maintenance,   // "LER_TeachingPos_Interface"
                           selectTeachingPos := 5,
                           indexTeachingPos := "HMI_Interface_Parameter".TeachingPosIndex,
                           configurationSetPositions := "Unit1.Em4.Config".cmAnodeMainPnP1AxisX.setPositions,
                           moduleInterface := "Unit1.Em4.HmiInterface".cmAnodeMainPnP1AxisX,
                           hmiInterface := "HMI_Interface_Parameter".TeachingPosInterface,
                           ENO => #_w1);
   "instTeachingPosAnodeMainPnP2AxisX"(EN := #_w1,   // "LER_TeachingPos_Interface"
                           enable := "Unit1.EmNodes".unitStatus.mode.maintenance,
                           selectTeachingPos := 6,
                           indexTeachingPos := "HMI_Interface_Parameter".TeachingPosIndex,
                           configurationSetPositions := "Unit1.Em4.Config".cmAnodeMainPnP2AxisX.setPositions,
                           moduleInterface := "Unit1.Em4.HmiInterface".cmAnodeMainPnP2AxisX,
                           hmiInterface := "HMI_Interface_Parameter".TeachingPosInterface,
                           ENO => #_w2);
   "instTeachingPosCathodeMainPnP1AxisX"(EN := #_w2,   // "LER_TeachingPos_Interface"
                           enable := "Unit1.EmNodes".unitStatus.mode.maintenance,
                           selectTeachingPos := 7,
                           indexTeachingPos := "HMI_Interface_Parameter".TeachingPosIndex,
                           configurationSetPositions := "Unit1.Em5.Config".cmCathodeMainPnP1AxisX.setPositions,
                           moduleInterface := "Unit1.Em5.HmiInterface".cmCathodeMainPnP1AxisX,
                           hmiInterface := "HMI_Interface_Parameter".TeachingPosInterface,
                           ENO => #_w3);
   IF #_w3 THEN
       "instTeachingPosCathodeMainPnP2AxisX"(enable := "Unit1.EmNodes".unitStatus.mode.maintenance,   // "LER_TeachingPos_Interface"
                               selectTeachingPos := 8,
                               indexTeachingPos := "HMI_Interface_Parameter".TeachingPosIndex,
                               configurationSetPositions := "Unit1.Em5.Config".cmCathodeMainPnP2AxisX.setPositions,
                               moduleInterface := "Unit1.Em5.HmiInterface".cmCathodeMainPnP2AxisX,
                               hmiInterface := "HMI_Interface_Parameter".TeachingPosInterface);
   END_IF;
END_REGION

REGION Network 19: Position Teaching (No 9~12)
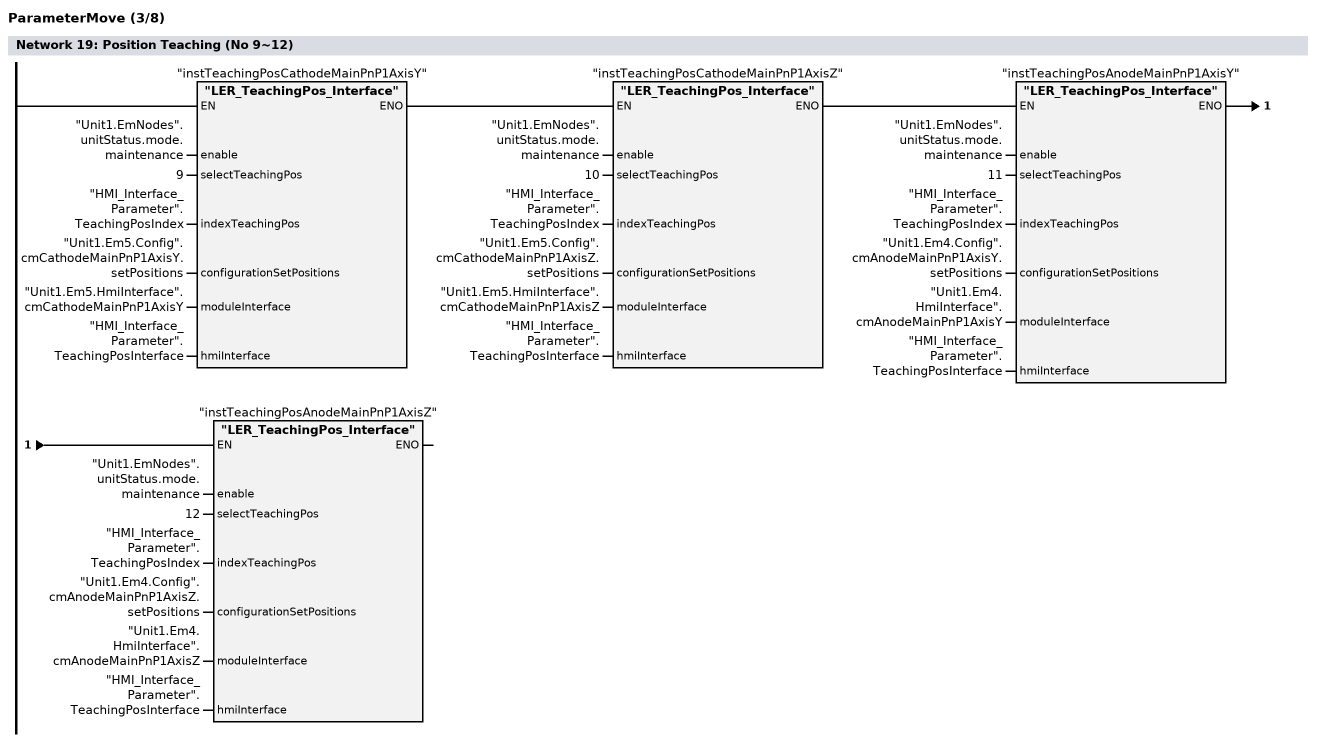
   RUNG wire#powerrail
      "instTeachingPosCathodeMainPnP1AxisY"(enable := "Unit1.EmNodes".unitStatus.mode.maintenance, selectTeachingPos := 9, indexTeachingPos := "HMI_Interface_Parameter".TeachingPosIndex, configurationSetPositions := "Unit1.Em5.Config".cmCathodeMainPnP1AxisY.setPositions, moduleInterface := "Unit1.Em5.HmiInterface".cmCathodeMainPnP1AxisY, hmiInterface := "HMI_Interface_Parameter".TeachingPosInterface)
      "instTeachingPosCathodeMainPnP1AxisZ"(enable := "Unit1.EmNodes".unitStatus.mode.maintenance, selectTeachingPos := 10, indexTeachingPos := "HMI_Interface_Parameter".TeachingPosIndex, configurationSetPositions := "Unit1.Em5.Config".cmCathodeMainPnP1AxisZ.setPositions, moduleInterface := "Unit1.Em5.HmiInterface".cmCathodeMainPnP1AxisZ, hmiInterface := "HMI_Interface_Parameter".TeachingPosInterface)
      "instTeachingPosAnodeMainPnP1AxisY"(enable := "Unit1.EmNodes".unitStatus.mode.maintenance, selectTeachingPos := 11, indexTeachingPos := "HMI_Interface_Parameter".TeachingPosIndex, configurationSetPositions := "Unit1.Em4.Config".cmAnodeMainPnP1AxisY.setPositions, moduleInterface := "Unit1.Em4.HmiInterface".cmAnodeMainPnP1AxisY, hmiInterface := "HMI_Interface_Parameter".TeachingPosInterface)
      "instTeachingPosAnodeMainPnP1AxisZ"(enable := "Unit1.EmNodes".unitStatus.mode.maintenance, selectTeachingPos := 12, indexTeachingPos := "HMI_Interface_Parameter".TeachingPosIndex, configurationSetPositions := "Unit1.Em4.Config".cmAnodeMainPnP1AxisZ.setPositions, moduleInterface := "Unit1.Em4.HmiInterface".cmAnodeMainPnP1AxisZ, hmiInterface := "HMI_Interface_Parameter".TeachingPosInterface)
   END_RUNG
   // the same network as SCL:
   "instTeachingPosCathodeMainPnP1AxisY"(enable := "Unit1.EmNodes".unitStatus.mode.maintenance,   // "LER_TeachingPos_Interface"
                           selectTeachingPos := 9,
                           indexTeachingPos := "HMI_Interface_Parameter".TeachingPosIndex,
                           configurationSetPositions := "Unit1.Em5.Config".cmCathodeMainPnP1AxisY.setPositions,
                           moduleInterface := "Unit1.Em5.HmiInterface".cmCathodeMainPnP1AxisY,
                           hmiInterface := "HMI_Interface_Parameter".TeachingPosInterface,
                           ENO => #_w1);
   "instTeachingPosCathodeMainPnP1AxisZ"(EN := #_w1,   // "LER_TeachingPos_Interface"
                           enable := "Unit1.EmNodes".unitStatus.mode.maintenance,
                           selectTeachingPos := 10,
                           indexTeachingPos := "HMI_Interface_Parameter".TeachingPosIndex,
                           configurationSetPositions := "Unit1.Em5.Config".cmCathodeMainPnP1AxisZ.setPositions,
                           moduleInterface := "Unit1.Em5.HmiInterface".cmCathodeMainPnP1AxisZ,
                           hmiInterface := "HMI_Interface_Parameter".TeachingPosInterface,
                           ENO => #_w2);
   "instTeachingPosAnodeMainPnP1AxisY"(EN := #_w2,   // "LER_TeachingPos_Interface"
                           enable := "Unit1.EmNodes".unitStatus.mode.maintenance,
                           selectTeachingPos := 11,
                           indexTeachingPos := "HMI_Interface_Parameter".TeachingPosIndex,
                           configurationSetPositions := "Unit1.Em4.Config".cmAnodeMainPnP1AxisY.setPositions,
                           moduleInterface := "Unit1.Em4.HmiInterface".cmAnodeMainPnP1AxisY,
                           hmiInterface := "HMI_Interface_Parameter".TeachingPosInterface,
                           ENO => #_w3);
   IF #_w3 THEN
       "instTeachingPosAnodeMainPnP1AxisZ"(enable := "Unit1.EmNodes".unitStatus.mode.maintenance,   // "LER_TeachingPos_Interface"
                               selectTeachingPos := 12,
                               indexTeachingPos := "HMI_Interface_Parameter".TeachingPosIndex,
                               configurationSetPositions := "Unit1.Em4.Config".cmAnodeMainPnP1AxisZ.setPositions,
                               moduleInterface := "Unit1.Em4.HmiInterface".cmAnodeMainPnP1AxisZ,
                               hmiInterface := "HMI_Interface_Parameter".TeachingPosInterface);
   END_IF;
END_REGION

REGION Network 20: Position Teaching (No 13~16)
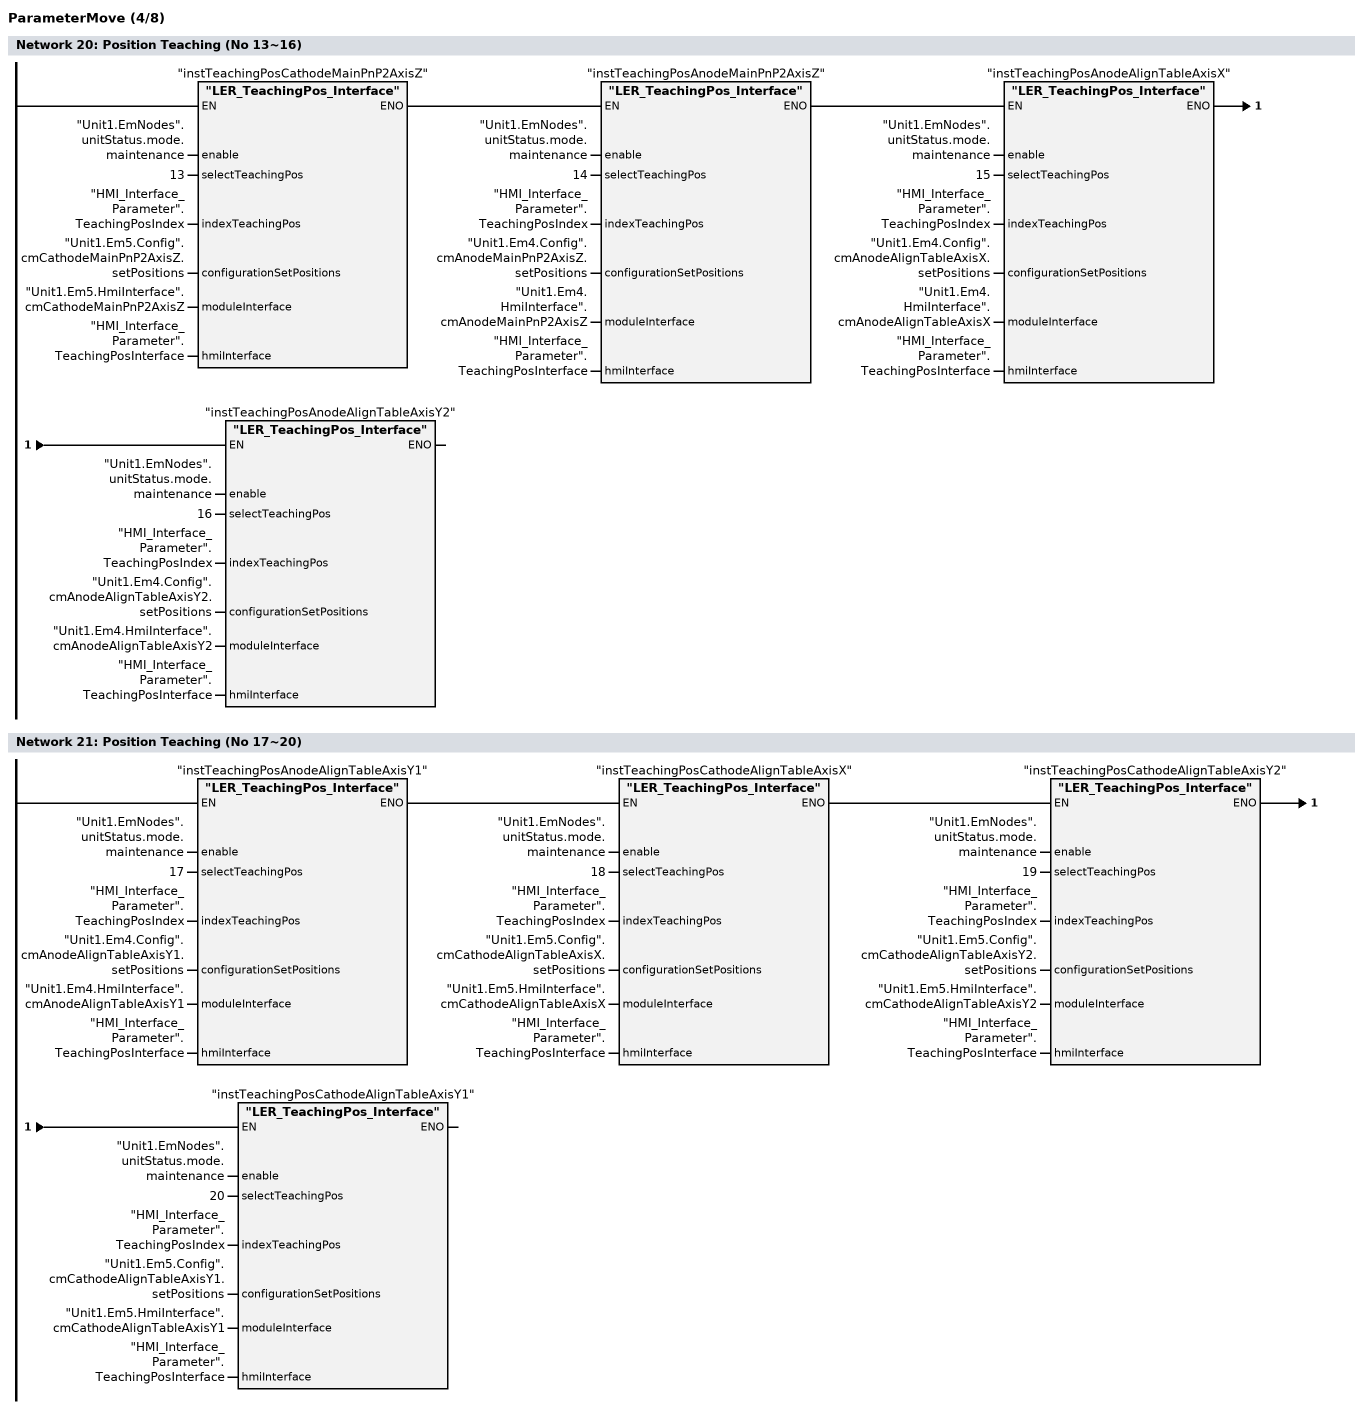
   RUNG wire#powerrail
      "instTeachingPosCathodeMainPnP2AxisZ"(enable := "Unit1.EmNodes".unitStatus.mode.maintenance, selectTeachingPos := 13, indexTeachingPos := "HMI_Interface_Parameter".TeachingPosIndex, configurationSetPositions := "Unit1.Em5.Config".cmCathodeMainPnP2AxisZ.setPositions, moduleInterface := "Unit1.Em5.HmiInterface".cmCathodeMainPnP2AxisZ, hmiInterface := "HMI_Interface_Parameter".TeachingPosInterface)
      "instTeachingPosAnodeMainPnP2AxisZ"(enable := "Unit1.EmNodes".unitStatus.mode.maintenance, selectTeachingPos := 14, indexTeachingPos := "HMI_Interface_Parameter".TeachingPosIndex, configurationSetPositions := "Unit1.Em4.Config".cmAnodeMainPnP2AxisZ.setPositions, moduleInterface := "Unit1.Em4.HmiInterface".cmAnodeMainPnP2AxisZ, hmiInterface := "HMI_Interface_Parameter".TeachingPosInterface)
      "instTeachingPosAnodeAlignTableAxisX"(enable := "Unit1.EmNodes".unitStatus.mode.maintenance, selectTeachingPos := 15, indexTeachingPos := "HMI_Interface_Parameter".TeachingPosIndex, configurationSetPositions := "Unit1.Em4.Config".cmAnodeAlignTableAxisX.setPositions, moduleInterface := "Unit1.Em4.HmiInterface".cmAnodeAlignTableAxisX, hmiInterface := "HMI_Interface_Parameter".TeachingPosInterface)
      "instTeachingPosAnodeAlignTableAxisY2"(enable := "Unit1.EmNodes".unitStatus.mode.maintenance, selectTeachingPos := 16, indexTeachingPos := "HMI_Interface_Parameter".TeachingPosIndex, configurationSetPositions := "Unit1.Em4.Config".cmAnodeAlignTableAxisY2.setPositions, moduleInterface := "Unit1.Em4.HmiInterface".cmAnodeAlignTableAxisY2, hmiInterface := "HMI_Interface_Parameter".TeachingPosInterface)
   END_RUNG
   // the same network as SCL:
   "instTeachingPosCathodeMainPnP2AxisZ"(enable := "Unit1.EmNodes".unitStatus.mode.maintenance,   // "LER_TeachingPos_Interface"
                           selectTeachingPos := 13,
                           indexTeachingPos := "HMI_Interface_Parameter".TeachingPosIndex,
                           configurationSetPositions := "Unit1.Em5.Config".cmCathodeMainPnP2AxisZ.setPositions,
                           moduleInterface := "Unit1.Em5.HmiInterface".cmCathodeMainPnP2AxisZ,
                           hmiInterface := "HMI_Interface_Parameter".TeachingPosInterface,
                           ENO => #_w1);
   "instTeachingPosAnodeMainPnP2AxisZ"(EN := #_w1,   // "LER_TeachingPos_Interface"
                           enable := "Unit1.EmNodes".unitStatus.mode.maintenance,
                           selectTeachingPos := 14,
                           indexTeachingPos := "HMI_Interface_Parameter".TeachingPosIndex,
                           configurationSetPositions := "Unit1.Em4.Config".cmAnodeMainPnP2AxisZ.setPositions,
                           moduleInterface := "Unit1.Em4.HmiInterface".cmAnodeMainPnP2AxisZ,
                           hmiInterface := "HMI_Interface_Parameter".TeachingPosInterface,
                           ENO => #_w2);
   "instTeachingPosAnodeAlignTableAxisX"(EN := #_w2,   // "LER_TeachingPos_Interface"
                           enable := "Unit1.EmNodes".unitStatus.mode.maintenance,
                           selectTeachingPos := 15,
                           indexTeachingPos := "HMI_Interface_Parameter".TeachingPosIndex,
                           configurationSetPositions := "Unit1.Em4.Config".cmAnodeAlignTableAxisX.setPositions,
                           moduleInterface := "Unit1.Em4.HmiInterface".cmAnodeAlignTableAxisX,
                           hmiInterface := "HMI_Interface_Parameter".TeachingPosInterface,
                           ENO => #_w3);
   IF #_w3 THEN
       "instTeachingPosAnodeAlignTableAxisY2"(enable := "Unit1.EmNodes".unitStatus.mode.maintenance,   // "LER_TeachingPos_Interface"
                               selectTeachingPos := 16,
                               indexTeachingPos := "HMI_Interface_Parameter".TeachingPosIndex,
                               configurationSetPositions := "Unit1.Em4.Config".cmAnodeAlignTableAxisY2.setPositions,
                               moduleInterface := "Unit1.Em4.HmiInterface".cmAnodeAlignTableAxisY2,
                               hmiInterface := "HMI_Interface_Parameter".TeachingPosInterface);
   END_IF;
END_REGION

REGION Network 21: Position Teaching (No 17~20)
   RUNG wire#powerrail
      "instTeachingPosAnodeAlignTableAxisY1"(enable := "Unit1.EmNodes".unitStatus.mode.maintenance, selectTeachingPos := 17, indexTeachingPos := "HMI_Interface_Parameter".TeachingPosIndex, configurationSetPositions := "Unit1.Em4.Config".cmAnodeAlignTableAxisY1.setPositions, moduleInterface := "Unit1.Em4.HmiInterface".cmAnodeAlignTableAxisY1, hmiInterface := "HMI_Interface_Parameter".TeachingPosInterface)
      "instTeachingPosCathodeAlignTableAxisX"(enable := "Unit1.EmNodes".unitStatus.mode.maintenance, selectTeachingPos := 18, indexTeachingPos := "HMI_Interface_Parameter".TeachingPosIndex, configurationSetPositions := "Unit1.Em5.Config".cmCathodeAlignTableAxisX.setPositions, moduleInterface := "Unit1.Em5.HmiInterface".cmCathodeAlignTableAxisX, hmiInterface := "HMI_Interface_Parameter".TeachingPosInterface)
      "instTeachingPosCathodeAlignTableAxisY2"(enable := "Unit1.EmNodes".unitStatus.mode.maintenance, selectTeachingPos := 19, indexTeachingPos := "HMI_Interface_Parameter".TeachingPosIndex, configurationSetPositions := "Unit1.Em5.Config".cmCathodeAlignTableAxisY2.setPositions, moduleInterface := "Unit1.Em5.HmiInterface".cmCathodeAlignTableAxisY2, hmiInterface := "HMI_Interface_Parameter".TeachingPosInterface)
      "instTeachingPosCathodeAlignTableAxisY1"(enable := "Unit1.EmNodes".unitStatus.mode.maintenance, selectTeachingPos := 20, indexTeachingPos := "HMI_Interface_Parameter".TeachingPosIndex, configurationSetPositions := "Unit1.Em5.Config".cmCathodeAlignTableAxisY1.setPositions, moduleInterface := "Unit1.Em5.HmiInterface".cmCathodeAlignTableAxisY1, hmiInterface := "HMI_Interface_Parameter".TeachingPosInterface)
   END_RUNG
   // the same network as SCL:
   "instTeachingPosAnodeAlignTableAxisY1"(enable := "Unit1.EmNodes".unitStatus.mode.maintenance,   // "LER_TeachingPos_Interface"
                           selectTeachingPos := 17,
                           indexTeachingPos := "HMI_Interface_Parameter".TeachingPosIndex,
                           configurationSetPositions := "Unit1.Em4.Config".cmAnodeAlignTableAxisY1.setPositions,
                           moduleInterface := "Unit1.Em4.HmiInterface".cmAnodeAlignTableAxisY1,
                           hmiInterface := "HMI_Interface_Parameter".TeachingPosInterface,
                           ENO => #_w1);
   "instTeachingPosCathodeAlignTableAxisX"(EN := #_w1,   // "LER_TeachingPos_Interface"
                           enable := "Unit1.EmNodes".unitStatus.mode.maintenance,
                           selectTeachingPos := 18,
                           indexTeachingPos := "HMI_Interface_Parameter".TeachingPosIndex,
                           configurationSetPositions := "Unit1.Em5.Config".cmCathodeAlignTableAxisX.setPositions,
                           moduleInterface := "Unit1.Em5.HmiInterface".cmCathodeAlignTableAxisX,
                           hmiInterface := "HMI_Interface_Parameter".TeachingPosInterface,
                           ENO => #_w2);
   "instTeachingPosCathodeAlignTableAxisY2"(EN := #_w2,   // "LER_TeachingPos_Interface"
                           enable := "Unit1.EmNodes".unitStatus.mode.maintenance,
                           selectTeachingPos := 19,
                           indexTeachingPos := "HMI_Interface_Parameter".TeachingPosIndex,
                           configurationSetPositions := "Unit1.Em5.Config".cmCathodeAlignTableAxisY2.setPositions,
                           moduleInterface := "Unit1.Em5.HmiInterface".cmCathodeAlignTableAxisY2,
                           hmiInterface := "HMI_Interface_Parameter".TeachingPosInterface,
                           ENO => #_w3);
   IF #_w3 THEN
       "instTeachingPosCathodeAlignTableAxisY1"(enable := "Unit1.EmNodes".unitStatus.mode.maintenance,   // "LER_TeachingPos_Interface"
                               selectTeachingPos := 20,
                               indexTeachingPos := "HMI_Interface_Parameter".TeachingPosIndex,
                               configurationSetPositions := "Unit1.Em5.Config".cmCathodeAlignTableAxisY1.setPositions,
                               moduleInterface := "Unit1.Em5.HmiInterface".cmCathodeAlignTableAxisY1,
                               hmiInterface := "HMI_Interface_Parameter".TeachingPosInterface);
   END_IF;
END_REGION

REGION Network 22: Position Teaching (No 21~24)
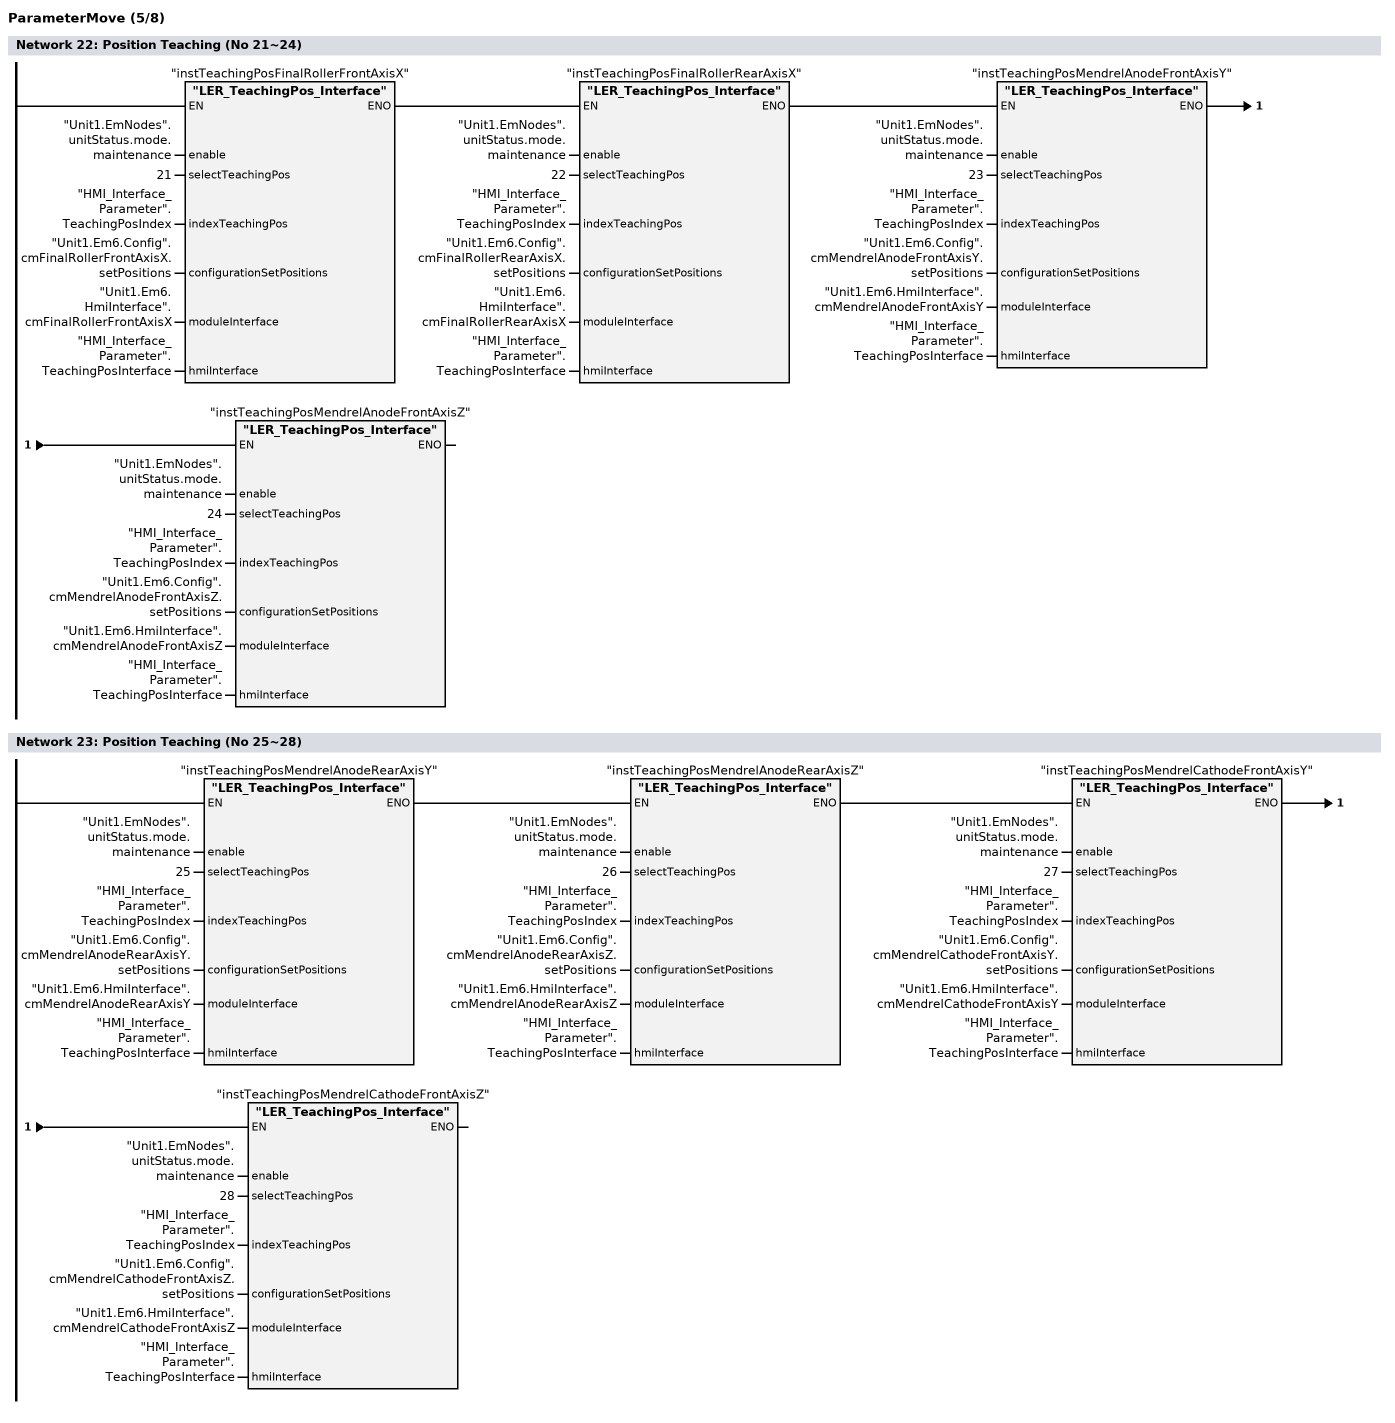
   RUNG wire#powerrail
      "instTeachingPosFinalRollerFrontAxisX"(enable := "Unit1.EmNodes".unitStatus.mode.maintenance, selectTeachingPos := 21, indexTeachingPos := "HMI_Interface_Parameter".TeachingPosIndex, configurationSetPositions := "Unit1.Em6.Config".cmFinalRollerFrontAxisX.setPositions, moduleInterface := "Unit1.Em6.HmiInterface".cmFinalRollerFrontAxisX, hmiInterface := "HMI_Interface_Parameter".TeachingPosInterface)
      "instTeachingPosFinalRollerRearAxisX"(enable := "Unit1.EmNodes".unitStatus.mode.maintenance, selectTeachingPos := 22, indexTeachingPos := "HMI_Interface_Parameter".TeachingPosIndex, configurationSetPositions := "Unit1.Em6.Config".cmFinalRollerRearAxisX.setPositions, moduleInterface := "Unit1.Em6.HmiInterface".cmFinalRollerRearAxisX, hmiInterface := "HMI_Interface_Parameter".TeachingPosInterface)
      "instTeachingPosMendrelAnodeFrontAxisY"(enable := "Unit1.EmNodes".unitStatus.mode.maintenance, selectTeachingPos := 23, indexTeachingPos := "HMI_Interface_Parameter".TeachingPosIndex, configurationSetPositions := "Unit1.Em6.Config".cmMendrelAnodeFrontAxisY.setPositions, moduleInterface := "Unit1.Em6.HmiInterface".cmMendrelAnodeFrontAxisY, hmiInterface := "HMI_Interface_Parameter".TeachingPosInterface)
      "instTeachingPosMendrelAnodeFrontAxisZ"(enable := "Unit1.EmNodes".unitStatus.mode.maintenance, selectTeachingPos := 24, indexTeachingPos := "HMI_Interface_Parameter".TeachingPosIndex, configurationSetPositions := "Unit1.Em6.Config".cmMendrelAnodeFrontAxisZ.setPositions, moduleInterface := "Unit1.Em6.HmiInterface".cmMendrelAnodeFrontAxisZ, hmiInterface := "HMI_Interface_Parameter".TeachingPosInterface)
   END_RUNG
   // the same network as SCL:
   "instTeachingPosFinalRollerFrontAxisX"(enable := "Unit1.EmNodes".unitStatus.mode.maintenance,   // "LER_TeachingPos_Interface"
                           selectTeachingPos := 21,
                           indexTeachingPos := "HMI_Interface_Parameter".TeachingPosIndex,
                           configurationSetPositions := "Unit1.Em6.Config".cmFinalRollerFrontAxisX.setPositions,
                           moduleInterface := "Unit1.Em6.HmiInterface".cmFinalRollerFrontAxisX,
                           hmiInterface := "HMI_Interface_Parameter".TeachingPosInterface,
                           ENO => #_w1);
   "instTeachingPosFinalRollerRearAxisX"(EN := #_w1,   // "LER_TeachingPos_Interface"
                           enable := "Unit1.EmNodes".unitStatus.mode.maintenance,
                           selectTeachingPos := 22,
                           indexTeachingPos := "HMI_Interface_Parameter".TeachingPosIndex,
                           configurationSetPositions := "Unit1.Em6.Config".cmFinalRollerRearAxisX.setPositions,
                           moduleInterface := "Unit1.Em6.HmiInterface".cmFinalRollerRearAxisX,
                           hmiInterface := "HMI_Interface_Parameter".TeachingPosInterface,
                           ENO => #_w2);
   "instTeachingPosMendrelAnodeFrontAxisY"(EN := #_w2,   // "LER_TeachingPos_Interface"
                           enable := "Unit1.EmNodes".unitStatus.mode.maintenance,
                           selectTeachingPos := 23,
                           indexTeachingPos := "HMI_Interface_Parameter".TeachingPosIndex,
                           configurationSetPositions := "Unit1.Em6.Config".cmMendrelAnodeFrontAxisY.setPositions,
                           moduleInterface := "Unit1.Em6.HmiInterface".cmMendrelAnodeFrontAxisY,
                           hmiInterface := "HMI_Interface_Parameter".TeachingPosInterface,
                           ENO => #_w3);
   IF #_w3 THEN
       "instTeachingPosMendrelAnodeFrontAxisZ"(enable := "Unit1.EmNodes".unitStatus.mode.maintenance,   // "LER_TeachingPos_Interface"
                               selectTeachingPos := 24,
                               indexTeachingPos := "HMI_Interface_Parameter".TeachingPosIndex,
                               configurationSetPositions := "Unit1.Em6.Config".cmMendrelAnodeFrontAxisZ.setPositions,
                               moduleInterface := "Unit1.Em6.HmiInterface".cmMendrelAnodeFrontAxisZ,
                               hmiInterface := "HMI_Interface_Parameter".TeachingPosInterface);
   END_IF;
END_REGION

REGION Network 23: Position Teaching (No 25~28)
   RUNG wire#powerrail
      "instTeachingPosMendrelAnodeRearAxisY"(enable := "Unit1.EmNodes".unitStatus.mode.maintenance, selectTeachingPos := 25, indexTeachingPos := "HMI_Interface_Parameter".TeachingPosIndex, configurationSetPositions := "Unit1.Em6.Config".cmMendrelAnodeRearAxisY.setPositions, moduleInterface := "Unit1.Em6.HmiInterface".cmMendrelAnodeRearAxisY, hmiInterface := "HMI_Interface_Parameter".TeachingPosInterface)
      "instTeachingPosMendrelAnodeRearAxisZ"(enable := "Unit1.EmNodes".unitStatus.mode.maintenance, selectTeachingPos := 26, indexTeachingPos := "HMI_Interface_Parameter".TeachingPosIndex, configurationSetPositions := "Unit1.Em6.Config".cmMendrelAnodeRearAxisZ.setPositions, moduleInterface := "Unit1.Em6.HmiInterface".cmMendrelAnodeRearAxisZ, hmiInterface := "HMI_Interface_Parameter".TeachingPosInterface)
      "instTeachingPosMendrelCathodeFrontAxisY"(enable := "Unit1.EmNodes".unitStatus.mode.maintenance, selectTeachingPos := 27, indexTeachingPos := "HMI_Interface_Parameter".TeachingPosIndex, configurationSetPositions := "Unit1.Em6.Config".cmMendrelCathodeFrontAxisY.setPositions, moduleInterface := "Unit1.Em6.HmiInterface".cmMendrelCathodeFrontAxisY, hmiInterface := "HMI_Interface_Parameter".TeachingPosInterface)
      "instTeachingPosMendrelCathodeFrontAxisZ"(enable := "Unit1.EmNodes".unitStatus.mode.maintenance, selectTeachingPos := 28, indexTeachingPos := "HMI_Interface_Parameter".TeachingPosIndex, configurationSetPositions := "Unit1.Em6.Config".cmMendrelCathodeFrontAxisZ.setPositions, moduleInterface := "Unit1.Em6.HmiInterface".cmMendrelCathodeFrontAxisZ, hmiInterface := "HMI_Interface_Parameter".TeachingPosInterface)
   END_RUNG
   // the same network as SCL:
   "instTeachingPosMendrelAnodeRearAxisY"(enable := "Unit1.EmNodes".unitStatus.mode.maintenance,   // "LER_TeachingPos_Interface"
                           selectTeachingPos := 25,
                           indexTeachingPos := "HMI_Interface_Parameter".TeachingPosIndex,
                           configurationSetPositions := "Unit1.Em6.Config".cmMendrelAnodeRearAxisY.setPositions,
                           moduleInterface := "Unit1.Em6.HmiInterface".cmMendrelAnodeRearAxisY,
                           hmiInterface := "HMI_Interface_Parameter".TeachingPosInterface,
                           ENO => #_w1);
   "instTeachingPosMendrelAnodeRearAxisZ"(EN := #_w1,   // "LER_TeachingPos_Interface"
                           enable := "Unit1.EmNodes".unitStatus.mode.maintenance,
                           selectTeachingPos := 26,
                           indexTeachingPos := "HMI_Interface_Parameter".TeachingPosIndex,
                           configurationSetPositions := "Unit1.Em6.Config".cmMendrelAnodeRearAxisZ.setPositions,
                           moduleInterface := "Unit1.Em6.HmiInterface".cmMendrelAnodeRearAxisZ,
                           hmiInterface := "HMI_Interface_Parameter".TeachingPosInterface,
                           ENO => #_w2);
   "instTeachingPosMendrelCathodeFrontAxisY"(EN := #_w2,   // "LER_TeachingPos_Interface"
                           enable := "Unit1.EmNodes".unitStatus.mode.maintenance,
                           selectTeachingPos := 27,
                           indexTeachingPos := "HMI_Interface_Parameter".TeachingPosIndex,
                           configurationSetPositions := "Unit1.Em6.Config".cmMendrelCathodeFrontAxisY.setPositions,
                           moduleInterface := "Unit1.Em6.HmiInterface".cmMendrelCathodeFrontAxisY,
                           hmiInterface := "HMI_Interface_Parameter".TeachingPosInterface,
                           ENO => #_w3);
   IF #_w3 THEN
       "instTeachingPosMendrelCathodeFrontAxisZ"(enable := "Unit1.EmNodes".unitStatus.mode.maintenance,   // "LER_TeachingPos_Interface"
                               selectTeachingPos := 28,
                               indexTeachingPos := "HMI_Interface_Parameter".TeachingPosIndex,
                               configurationSetPositions := "Unit1.Em6.Config".cmMendrelCathodeFrontAxisZ.setPositions,
                               moduleInterface := "Unit1.Em6.HmiInterface".cmMendrelCathodeFrontAxisZ,
                               hmiInterface := "HMI_Interface_Parameter".TeachingPosInterface);
   END_IF;
END_REGION

